# B&R Automation Studio project PLC code - cp (part 21)

#### PLC2Kernel_AutoCode.st
```iecst
// THIS CODE IS AUTOGENERATED. DO NOT MODIFY IT WITH AUTOMATION STUDIO
// Generation: 10/07/2024 16:17:34
// Program version: 2.1.4.0

ACTION PLC2Kernel_AutoCode:
HoldingRegister[1000]:=gPLC.iVarsVersion0;
HoldingRegister[1001]:=gPLC.iVarsVersion1;
HoldingRegister[1002]:=gPLC.iVarsVersion2;
HoldingRegister[1003]:=gPLC.iVersion0;
HoldingRegister[1004]:=gPLC.iVersion1;
HoldingRegister[1005]:=gPLC.iVersion2;
HoldingRegister[1006]:=gPLC.iVersion3;
HoldingRegister[1007].0:=gMachine.Al.Alarm.xAlr24Vdc;
HoldingRegister[1007].1:=gTransVacuum[1].parSw.xActiveOutOfProduction;
HoldingRegister[1007].2:=gTransVacuum[1].Status.xStartedMan;
HoldingRegister[1007].3:=gInks[1].parSw.xActTestMode;
HoldingRegister[1007].4:=gInks[2].parSw.xActTestMode;
HoldingRegister[1007].5:=gInks[3].parSw.xActTestMode;
HoldingRegister[1007].6:=gInks[4].parSw.xActTestMode;
HoldingRegister[1007].7:=gInks[5].parSw.xActTestMode;
HoldingRegister[1007].8:=gInks[6].parSw.xActTestMode;
HoldingRegister[1007].9:=gInks[7].parSw.xActTestMode;
HoldingRegister[1007].10:=gInks[8].parSw.xActTestMode;
HoldingRegister[1007].11:=gInks[9].parSw.xActTestMode;
HoldingRegister[1007].12:=gInks[10].parSw.xActTestMode;
HoldingRegister[1007].13:=gInks[11].parSw.xActTestMode;
HoldingRegister[1007].14:=gInks[12].parSw.xActTestMode;
HoldingRegister[1007].15:=gMachine.Al.Alarm.xAlarmAir1;
HoldingRegister[1008].0:=gBlock[1].Al.xAlAirVenturi;
HoldingRegister[1008].1:=gBlock[2].Al.xAlAirVenturi;
HoldingRegister[1008].2:=gMachine.Al.Alarm.xNotLoadedImage;
HoldingRegister[1008].4:=gMachine.St.Mode.xAuto;
HoldingRegister[1008].5:=gBlock[1].Al.xAlrRearSafety;
HoldingRegister[1008].6:=gBlock[2].Al.xAlrRearSafety;
HoldingRegister[1008].7:=gBlock[1].Al.xAlrDecreaseCleanOffset;
HoldingRegister[1008].8:=gBlock[2].Al.xAlrDecreaseCleanOffset;
HoldingRegister[1008].9:=gInks[1].status.xEnabledBarToPrint;
HoldingRegister[1008].10:=gInks[2].status.xEnabledBarToPrint;
HoldingRegister[1008].11:=gInks[3].status.xEnabledBarToPrint;
HoldingRegister[1008].12:=gInks[4].status.xEnabledBarToPrint;
HoldingRegister[1008].13:=gInks[5].status.xEnabledBarToPrint;
HoldingRegister[1008].14:=gInks[6].status.xEnabledBarToPrint;
HoldingRegister[1008].15:=gInks[7].status.xEnabledBarToPrint;
HoldingRegister[1009].0:=gInks[8].status.xEnabledBarToPrint;
HoldingRegister[1009].1:=gInks[9].status.xEnabledBarToPrint;
HoldingRegister[1009].2:=gInks[10].status.xEnabledBarToPrint;
HoldingRegister[1009].3:=gInks[11].status.xEnabledBarToPrint;
HoldingRegister[1009].4:=gInks[12].status.xEnabledBarToPrint;
HoldingRegister[1009].5:=gMachine.Al.Alarm.xAlarmNotInPrintPosition;
HoldingRegister[1009].6:=gBlock[1].Al.xAlrFrontCurtain;
HoldingRegister[1009].7:=gBlock[2].Al.xAlrFrontCurtain;
HoldingRegister[1009].10:=gBelt.Al.xControllerNotReady;
HoldingRegister[1009].11:=gThicknessCtrl.status.Belt.xBeltEmpty;
HoldingRegister[1009].13:=gBlock[1].Al.xSiUnitPowerOff;
HoldingRegister[1009].14:=gBlock[2].Al.xSiUnitPowerOff;
HoldingRegister[1009].15:=gTransVacuum[1].Alarms.xAlrVacuumSensor;
HoldingRegister[1010].0:=gTransVacuum[2].Alarms.xAlrVacuumSensor;
HoldingRegister[1010].1:=gBlock[1].Al.xAlrDriveProtection;
HoldingRegister[1010].2:=gBlock[2].Al.xAlrDriveProtection;
HoldingRegister[1010].3:=gInks[1].Al.xAlrBrokenMeniscus;
HoldingRegister[1010].4:=gInks[2].Al.xAlrBrokenMeniscus;
HoldingRegister[1010].5:=gInks[3].Al.xAlrBrokenMeniscus;
HoldingRegister[1010].6:=gInks[4].Al.xAlrBrokenMeniscus;
HoldingRegister[1010].7:=gInks[5].Al.xAlrBrokenMeniscus;
HoldingRegister[1010].8:=gInks[6].Al.xAlrBrokenMeniscus;
HoldingRegister[1010].9:=gInks[7].Al.xAlrBrokenMeniscus;
HoldingRegister[1010].10:=gInks[8].Al.xAlrBrokenMeniscus;
HoldingRegister[1010].11:=gInks[9].Al.xAlrBrokenMeniscus;
HoldingRegister[1010].12:=gInks[10].Al.xAlrBrokenMeniscus;
HoldingRegister[1010].13:=gInks[11].Al.xAlrBrokenMeniscus;
HoldingRegister[1010].14:=gInks[12].Al.xAlrBrokenMeniscus;
HoldingRegister[1010].15:=gChiller[1].Alarm.xCheckChiller;
HoldingRegister[1011].0:=gBlock[1].Al.xAlrCheckHomingSensor;
HoldingRegister[1011].1:=gBlock[2].Al.xAlrCheckHomingSensor;
HoldingRegister[1011].2:=gChiller[1].Alarm.xInAlarm;
HoldingRegister[1011].3:=gChiller[1].Alarm.xNotRunning;
HoldingRegister[1011].4:=gMachine.parSw.Clean.xCleaningBlocksInSeq;
HoldingRegister[1011].5:=gBlock[1].Al.xCleanMotorControllerNotReady;
HoldingRegister[1011].6:=gBlock[2].Al.xCleanMotorControllerNotReady;
HoldingRegister[1011].7:=gBelt.Al.xAlrComDrive;
HoldingRegister[1011].8:=gBlock[1].Al.xAlrComBarMtr;
HoldingRegister[1011].9:=gBlock[2].Al.xAlrComBarMtr;
HoldingRegister[1011].10:=gBlock[1].Al.xAlrComCleanMtr;
HoldingRegister[1011].11:=gBlock[2].Al.xAlrComCleanMtr;
HoldingRegister[1011].12:=gBlock[1].Al.xAlrComSiUnit;
HoldingRegister[1011].13:=gBlock[2].Al.xAlrComSiUnit;
HoldingRegister[1012].0:=gTransVacuum[1].Alarms.xAlrComsBlower;
HoldingRegister[1012].1:=gNonCrash[1].Alarms.xAlrComsDrive;
HoldingRegister[1012].2:=gTransVacuum[2].Alarms.xAlrComsBlower;
HoldingRegister[1012].3:=gMachine.Al.Alarm.xAlarmComPcPLC;
HoldingRegister[1012].4:=gPhotoCells.Alarms.xComsMotorError;
HoldingRegister[1012].7:=gMachine.St.Consent.xConsent;
HoldingRegister[1012].8:=gPhotoCells.Alarms.xContinuousActPDPhcell;
HoldingRegister[1012].9:=gMachine.Pt.xControlledByLine;
HoldingRegister[1012].10:=gBlock[1].Al.xAlrControllerNotReady;
HoldingRegister[1012].11:=gBlock[2].Al.xAlrControllerNotReady;
HoldingRegister[1012].12:=gNonCrash[1].Alarms.xControllerNotReady;
HoldingRegister[1012].13:=gBlock[1].Al.xAlrBlockReachedMaxPosition;
HoldingRegister[1012].14:=gBlock[2].Al.xAlrBlockReachedMaxPosition;
HoldingRegister[1012].15:=gInks[1].Al.xAlrTankToFillIn;
HoldingRegister[1013].0:=gInks[2].Al.xAlrTankToFillIn;
HoldingRegister[1013].1:=gInks[3].Al.xAlrTankToFillIn;
HoldingRegister[1013].2:=gInks[4].Al.xAlrTankToFillIn;
HoldingRegister[1013].3:=gInks[5].Al.xAlrTankToFillIn;
HoldingRegister[1013].4:=gInks[6].Al.xAlrTankToFillIn;
HoldingRegister[1013].5:=gInks[7].Al.xAlrTankToFillIn;
HoldingRegister[1013].6:=gInks[8].Al.xAlrTankToFillIn;
HoldingRegister[1013].7:=gInks[9].Al.xAlrTankToFillIn;
HoldingRegister[1013].8:=gInks[10].Al.xAlrTankToFillIn;
HoldingRegister[1013].9:=gInks[11].Al.xAlrTankToFillIn;
HoldingRegister[1013].10:=gInks[12].Al.xAlrTankToFillIn;
HoldingRegister[1013].11:=gInks[1].Al.xAlrTankEmpty;
HoldingRegister[1013].12:=gInks[2].Al.xAlrTankEmpty;
HoldingRegister[1013].13:=gInks[3].Al.xAlrTankEmpty;
HoldingRegister[1013].14:=gInks[4].Al.xAlrTankEmpty;
HoldingRegister[1013].15:=gInks[5].Al.xAlrTankEmpty;
HoldingRegister[1014].0:=gInks[6].Al.xAlrTankEmpty;
HoldingRegister[1014].1:=gInks[7].Al.xAlrTankEmpty;
HoldingRegister[1014].2:=gInks[8].Al.xAlrTankEmpty;
HoldingRegister[1014].3:=gInks[9].Al.xAlrTankEmpty;
HoldingRegister[1014].4:=gInks[10].Al.xAlrTankEmpty;
HoldingRegister[1014].5:=gInks[11].Al.xAlrTankEmpty;
HoldingRegister[1014].6:=gInks[12].Al.xAlrTankEmpty;
HoldingRegister[1014].7:=gInks[1].Al.xAlrDiffInCtrlTempTank;
HoldingRegister[1014].8:=gInks[2].Al.xAlrDiffInCtrlTempTank;
HoldingRegister[1014].9:=gInks[3].Al.xAlrDiffInCtrlTempTank;
HoldingRegister[1014].10:=gInks[4].Al.xAlrDiffInCtrlTempTank;
HoldingRegister[1014].11:=gInks[5].Al.xAlrDiffInCtrlTempTank;
HoldingRegister[1014].12:=gInks[6].Al.xAlrDiffInCtrlTempTank;
HoldingRegister[1014].13:=gInks[7].Al.xAlrDiffInCtrlTempTank;
HoldingRegister[1014].14:=gInks[8].Al.xAlrDiffInCtrlTempTank;
HoldingRegister[1014].15:=gInks[9].Al.xAlrDiffInCtrlTempTank;
HoldingRegister[1015].0:=gInks[10].Al.xAlrDiffInCtrlTempTank;
HoldingRegister[1015].1:=gInks[11].Al.xAlrDiffInCtrlTempTank;
HoldingRegister[1015].2:=gInks[12].Al.xAlrDiffInCtrlTempTank;
HoldingRegister[1015].3:=gInks[1].Al.xAlrDiffInCtrlTemp;
HoldingRegister[1015].4:=gInks[2].Al.xAlrDiffInCtrlTemp;
HoldingRegister[1015].5:=gInks[3].Al.xAlrDiffInCtrlTemp;
HoldingRegister[1015].6:=gInks[4].Al.xAlrDiffInCtrlTemp;
HoldingRegister[1015].7:=gInks[5].Al.xAlrDiffInCtrlTemp;
HoldingRegister[1015].8:=gInks[6].Al.xAlrDiffInCtrlTemp;
HoldingRegister[1015].9:=gInks[7].Al.xAlrDiffInCtrlTemp;
HoldingRegister[1015].10:=gInks[8].Al.xAlrDiffInCtrlTemp;
HoldingRegister[1015].11:=gInks[9].Al.xAlrDiffInCtrlTemp;
HoldingRegister[1015].12:=gInks[10].Al.xAlrDiffInCtrlTemp;
HoldingRegister[1015].13:=gInks[11].Al.xAlrDiffInCtrlTemp;
HoldingRegister[1015].14:=gInks[12].Al.xAlrDiffInCtrlTemp;
HoldingRegister[1015].15:=gBlock[1].Al.xAlrDif;
HoldingRegister[1016].0:=gBlock[2].Al.xAlrDif;
HoldingRegister[1016].2:=gNonCrash[1].Alarms.xAlrDiffContact;
HoldingRegister[1016].3:=gInks[1].Al.xAlrDifCtrlTempExcessive;
HoldingRegister[1016].4:=gInks[2].Al.xAlrDifCtrlTempExcessive;
HoldingRegister[1016].5:=gInks[3].Al.xAlrDifCtrlTempExcessive;
HoldingRegister[1016].6:=gInks[4].Al.xAlrDifCtrlTempExcessive;
HoldingRegister[1016].7:=gInks[5].Al.xAlrDifCtrlTempExcessive;
HoldingRegister[1016].8:=gInks[6].Al.xAlrDifCtrlTempExcessive;
HoldingRegister[1016].9:=gInks[7].Al.xAlrDifCtrlTempExcessive;
HoldingRegister[1016].10:=gInks[8].Al.xAlrDifCtrlTempExcessive;
HoldingRegister[1016].11:=gInks[9].Al.xAlrDifCtrlTempExcessive;
HoldingRegister[1016].12:=gInks[10].Al.xAlrDifCtrlTempExcessive;
HoldingRegister[1016].13:=gInks[11].Al.xAlrDifCtrlTempExcessive;
HoldingRegister[1016].14:=gInks[12].Al.xAlrDifCtrlTempExcessive;
HoldingRegister[1016].15:=gInks[1].Al.xAlrDiffVacuum;
HoldingRegister[1017].0:=gInks[2].Al.xAlrDiffVacuum;
HoldingRegister[1017].1:=gInks[3].Al.xAlrDiffVacuum;
HoldingRegister[1017].2:=gInks[4].Al.xAlrDiffVacuum;
HoldingRegister[1017].3:=gInks[5].Al.xAlrDiffVacuum;
HoldingRegister[1017].4:=gInks[6].Al.xAlrDiffVacuum;
HoldingRegister[1017].5:=gInks[7].Al.xAlrDiffVacuum;
HoldingRegister[1017].6:=gInks[8].Al.xAlrDiffVacuum;
HoldingRegister[1017].7:=gInks[9].Al.xAlrDiffVacuum;
HoldingRegister[1017].8:=gInks[10].Al.xAlrDiffVacuum;
HoldingRegister[1017].9:=gInks[11].Al.xAlrDiffVacuum;
HoldingRegister[1017].10:=gInks[12].Al.xAlrDiffVacuum;
HoldingRegister[1017].11:=gDing.Alarms.xAlDingNoDigLaserSensor;
HoldingRegister[1017].12:=gMachine.parSw.Dtp.xDoubleLine;
HoldingRegister[1017].13:=gMachine.St.xDoubleLineAllowed;
HoldingRegister[1017].14:=gBlock[1].Al.xAlrFrontEmergencyStop;
HoldingRegister[1017].15:=gBlock[2].Al.xAlrFrontEmergencyStop;
HoldingRegister[1018].0:=gBlock[1].Al.xAlrFrontSafetyCircuit;
HoldingRegister[1018].1:=gBlock[2].Al.xAlrFrontSafetyCircuit;
HoldingRegister[1018].2:=gBlock[1].Al.xAlrRearEmergencyStop;
HoldingRegister[1018].3:=gBlock[2].Al.xAlrRearEmergencyStop;
HoldingRegister[1018].4:=gBlock[1].Al.xAlrRearSafetyCircuit;
HoldingRegister[1018].5:=gBlock[2].Al.xAlrRearSafetyCircuit;
HoldingRegister[1018].6:=gBlock[1].Status.xIsWaterBlock;
HoldingRegister[1018].7:=gBlock[2].Status.xIsWaterBlock;
HoldingRegister[1018].9:=gJamDetect[1].Parameters.xJamEnabled;
HoldingRegister[1018].10:=gNonCrash[1].Status.xEnabled;
HoldingRegister[1018].11:=gMachine.parSw.Clean.xEnableCleaningInStopMode;
HoldingRegister[1018].12:=gBlock[1].parSw.xEnableToMovements;
HoldingRegister[1018].13:=gBlock[2].parSw.xEnableToMovements;
HoldingRegister[1018].14:=gBlock[1].Al.xAlrEnabCleanMtrDiffLvL;
HoldingRegister[1018].15:=gBlock[2].Al.xAlrEnabCleanMtrDiffLvL;
HoldingRegister[1019].0:=gInks[1].parSw.Temp.xTankHeaterEnabled;
HoldingRegister[1019].1:=gInks[2].parSw.Temp.xTankHeaterEnabled;
HoldingRegister[1019].2:=gInks[3].parSw.Temp.xTankHeaterEnabled;
HoldingRegister[1019].3:=gInks[4].parSw.Temp.xTankHeaterEnabled;
HoldingRegister[1019].4:=gInks[5].parSw.Temp.xTankHeaterEnabled;
HoldingRegister[1019].5:=gInks[6].parSw.Temp.xTankHeaterEnabled;
HoldingRegister[1019].6:=gInks[7].parSw.Temp.xTankHeaterEnabled;
HoldingRegister[1019].7:=gInks[8].parSw.Temp.xTankHeaterEnabled;
HoldingRegister[1019].8:=gInks[9].parSw.Temp.xTankHeaterEnabled;
HoldingRegister[1019].9:=gInks[10].parSw.Temp.xTankHeaterEnabled;
HoldingRegister[1019].10:=gInks[11].parSw.Temp.xTankHeaterEnabled;
HoldingRegister[1019].11:=gInks[12].parSw.Temp.xTankHeaterEnabled;
HoldingRegister[1019].12:=gBlock[1].parSw.xEnableToPrint;
HoldingRegister[1019].13:=gBlock[2].parSw.xEnableToPrint;
HoldingRegister[1019].14:=gChiller[1].Alarm.xAlrEnvTempSensBrokn;
HoldingRegister[1019].15:=gTransVacuum[1].Alarms.xAlrDriveBlowerError;
HoldingRegister[1020].0:=gNonCrash[1].Alarms.xAlrDriveError;
HoldingRegister[1020].1:=gPhotoCells.Alarms.xMotorError;
HoldingRegister[1020].2:=gTransVacuum[2].Alarms.xAlrDriveBlowerError;
HoldingRegister[1020].3:=gMachine.parSw.Electronics.xPrintServerOK;
HoldingRegister[1020].4:=gMachine.parSw.Electronics.xRobotReadyL1;
HoldingRegister[1020].5:=gMachine.parSw.Electronics.xRobotReadyL2;
HoldingRegister[1020].6:=gInks[1].Al.xAlrVacuumSensor1;
HoldingRegister[1020].7:=gInks[2].Al.xAlrVacuumSensor1;
HoldingRegister[1020].8:=gInks[3].Al.xAlrVacuumSensor1;
HoldingRegister[1020].9:=gInks[4].Al.xAlrVacuumSensor1;
HoldingRegister[1020].10:=gInks[5].Al.xAlrVacuumSensor1;
HoldingRegister[1020].11:=gInks[6].Al.xAlrVacuumSensor1;
HoldingRegister[1020].12:=gInks[7].Al.xAlrVacuumSensor1;
HoldingRegister[1020].13:=gInks[8].Al.xAlrVacuumSensor1;
HoldingRegister[1020].14:=gInks[9].Al.xAlrVacuumSensor1;
HoldingRegister[1020].15:=gInks[10].Al.xAlrVacuumSensor1;
HoldingRegister[1021].0:=gInks[11].Al.xAlrVacuumSensor1;
HoldingRegister[1021].1:=gInks[12].Al.xAlrVacuumSensor1;
HoldingRegister[1021].2:=gInks[1].Al.xAlrVacuumSensor2;
HoldingRegister[1021].3:=gInks[2].Al.xAlrVacuumSensor2;
HoldingRegister[1021].4:=gInks[3].Al.xAlrVacuumSensor2;
HoldingRegister[1021].5:=gInks[4].Al.xAlrVacuumSensor2;
HoldingRegister[1021].6:=gInks[5].Al.xAlrVacuumSensor2;
HoldingRegister[1021].7:=gInks[6].Al.xAlrVacuumSensor2;
HoldingRegister[1021].8:=gInks[7].Al.xAlrVacuumSensor2;
HoldingRegister[1021].9:=gInks[8].Al.xAlrVacuumSensor2;
HoldingRegister[1021].10:=gInks[9].Al.xAlrVacuumSensor2;
HoldingRegister[1021].11:=gInks[10].Al.xAlrVacuumSensor2;
HoldingRegister[1021].12:=gInks[11].Al.xAlrVacuumSensor2;
HoldingRegister[1021].13:=gInks[12].Al.xAlrVacuumSensor2;
HoldingRegister[1021].14:=gBelt.Al.xAlrPowerBeltError;
HoldingRegister[1021].15:=gBlock[1].Al.xAlrFrontSafety;
HoldingRegister[1022].0:=gBlock[2].Al.xAlrFrontSafety;
HoldingRegister[1022].1:=gTransVacuum[1].Alarms.xAlrJointSystemPressure;
HoldingRegister[1022].2:=gMachine.parSw.CleanBelt.xCleanBeltByTiles;
HoldingRegister[1022].3:=gMachine.parSw.CleanBelt.xCleanBeltByTime;
HoldingRegister[1022].4:=gMachine.parSw.CleanBeltTop.xCleanBeltByTiles;
HoldingRegister[1022].5:=gMachine.parSw.CleanBeltTop.xCleanBeltByTime;
HoldingRegister[1022].6:=gMachine.Al.Alarm.xAlarmEnableWithoutBarsOn;
HoldingRegister[1022].7:=gInks[1].Al.xAlrHeaterOutFault;
HoldingRegister[1022].8:=gInks[2].Al.xAlrHeaterOutFault;
HoldingRegister[1022].9:=gInks[3].Al.xAlrHeaterOutFault;
HoldingRegister[1022].10:=gInks[4].Al.xAlrHeaterOutFault;
HoldingRegister[1022].11:=gInks[5].Al.xAlrHeaterOutFault;
HoldingRegister[1022].12:=gInks[6].Al.xAlrHeaterOutFault;
HoldingRegister[1022].13:=gInks[7].Al.xAlrHeaterOutFault;
HoldingRegister[1022].14:=gInks[8].Al.xAlrHeaterOutFault;
HoldingRegister[1022].15:=gInks[9].Al.xAlrHeaterOutFault;
HoldingRegister[1023].0:=gInks[10].Al.xAlrHeaterOutFault;
HoldingRegister[1023].1:=gInks[11].Al.xAlrHeaterOutFault;
HoldingRegister[1023].2:=gInks[12].Al.xAlrHeaterOutFault;
HoldingRegister[1023].3:=gInks[1].Al.xAlrHeaterReachsMaxTemp;
HoldingRegister[1023].4:=gInks[2].Al.xAlrHeaterReachsMaxTemp;
HoldingRegister[1023].5:=gInks[3].Al.xAlrHeaterReachsMaxTemp;
HoldingRegister[1023].6:=gInks[4].Al.xAlrHeaterReachsMaxTemp;
HoldingRegister[1023].7:=gInks[5].Al.xAlrHeaterReachsMaxTemp;
HoldingRegister[1023].8:=gInks[6].Al.xAlrHeaterReachsMaxTemp;
HoldingRegister[1023].9:=gInks[7].Al.xAlrHeaterReachsMaxTemp;
HoldingRegister[1023].10:=gInks[8].Al.xAlrHeaterReachsMaxTemp;
HoldingRegister[1023].11:=gInks[9].Al.xAlrHeaterReachsMaxTemp;
HoldingRegister[1023].12:=gInks[10].Al.xAlrHeaterReachsMaxTemp;
HoldingRegister[1023].13:=gInks[11].Al.xAlrHeaterReachsMaxTemp;
HoldingRegister[1023].14:=gInks[12].Al.xAlrHeaterReachsMaxTemp;
HoldingRegister[1023].15:=gInks[1].Al.xAlrHeaterTankReachsMaxTemp;
HoldingRegister[1024].0:=gInks[2].Al.xAlrHeaterTankReachsMaxTemp;
HoldingRegister[1024].1:=gInks[3].Al.xAlrHeaterTankReachsMaxTemp;
HoldingRegister[1024].2:=gInks[4].Al.xAlrHeaterTankReachsMaxTemp;
HoldingRegister[1024].3:=gInks[5].Al.xAlrHeaterTankReachsMaxTemp;
HoldingRegister[1024].4:=gInks[6].Al.xAlrHeaterTankReachsMaxTemp;
HoldingRegister[1024].5:=gInks[7].Al.xAlrHeaterTankReachsMaxTemp;
HoldingRegister[1024].6:=gInks[8].Al.xAlrHeaterTankReachsMaxTemp;
HoldingRegister[1024].7:=gInks[9].Al.xAlrHeaterTankReachsMaxTemp;
HoldingRegister[1024].8:=gInks[10].Al.xAlrHeaterTankReachsMaxTemp;
HoldingRegister[1024].9:=gInks[11].Al.xAlrHeaterTankReachsMaxTemp;
HoldingRegister[1024].10:=gInks[12].Al.xAlrHeaterTankReachsMaxTemp;
HoldingRegister[1024].11:=gBelt.Al.xAlrProtDrive;
HoldingRegister[1024].12:=gBlock[1].Al.xAlrCleanMtrNoRef;
HoldingRegister[1024].13:=gBlock[2].Al.xAlrCleanMtrNoRef;
HoldingRegister[1024].14:=gBlock[1].Status.Icla.xHomed;
HoldingRegister[1024].15:=gBlock[2].Status.Icla.xHomed;
HoldingRegister[1025].0:=gMachine.Al.Warning.xNotLoadedImage;
HoldingRegister[1025].1:=gInks[1].Al.xAlrLevelSensorError;
HoldingRegister[1025].2:=gInks[2].Al.xAlrLevelSensorError;
HoldingRegister[1025].3:=gInks[3].Al.xAlrLevelSensorError;
HoldingRegister[1025].4:=gInks[4].Al.xAlrLevelSensorError;
HoldingRegister[1025].5:=gInks[5].Al.xAlrLevelSensorError;
HoldingRegister[1025].6:=gInks[6].Al.xAlrLevelSensorError;
HoldingRegister[1025].7:=gInks[7].Al.xAlrLevelSensorError;
HoldingRegister[1025].8:=gInks[8].Al.xAlrLevelSensorError;
HoldingRegister[1025].9:=gInks[9].Al.xAlrLevelSensorError;
HoldingRegister[1025].10:=gInks[10].Al.xAlrLevelSensorError;
HoldingRegister[1025].11:=gInks[11].Al.xAlrLevelSensorError;
HoldingRegister[1025].12:=gInks[12].Al.xAlrLevelSensorError;
HoldingRegister[1025].13:=gInks[1].Al.xAlrIncoherTempHeat;
HoldingRegister[1025].14:=gInks[2].Al.xAlrIncoherTempHeat;
HoldingRegister[1025].15:=gInks[3].Al.xAlrIncoherTempHeat;
HoldingRegister[1026].0:=gInks[4].Al.xAlrIncoherTempHeat;
HoldingRegister[1026].1:=gInks[5].Al.xAlrIncoherTempHeat;
HoldingRegister[1026].2:=gInks[6].Al.xAlrIncoherTempHeat;
HoldingRegister[1026].3:=gInks[7].Al.xAlrIncoherTempHeat;
HoldingRegister[1026].4:=gInks[8].Al.xAlrIncoherTempHeat;
HoldingRegister[1026].5:=gInks[9].Al.xAlrIncoherTempHeat;
HoldingRegister[1026].6:=gInks[10].Al.xAlrIncoherTempHeat;
HoldingRegister[1026].7:=gInks[11].Al.xAlrIncoherTempHeat;
HoldingRegister[1026].8:=gInks[12].Al.xAlrIncoherTempHeat;
HoldingRegister[1026].9:=gPhotoCells.Alarms.xIncoherPhotocellSystem;
HoldingRegister[1026].10:=gBlock[1].Al.xAlrIncoherPositCleanMtr;
HoldingRegister[1026].11:=gBlock[2].Al.xAlrIncoherPositCleanMtr;
HoldingRegister[1026].12:=gInks[1].Al.xAlrIncoherTempTank;
HoldingRegister[1026].13:=gInks[2].Al.xAlrIncoherTempTank;
HoldingRegister[1026].14:=gInks[3].Al.xAlrIncoherTempTank;
HoldingRegister[1026].15:=gInks[4].Al.xAlrIncoherTempTank;
HoldingRegister[1027].0:=gInks[5].Al.xAlrIncoherTempTank;
HoldingRegister[1027].1:=gInks[6].Al.xAlrIncoherTempTank;
HoldingRegister[1027].2:=gInks[7].Al.xAlrIncoherTempTank;
HoldingRegister[1027].3:=gInks[8].Al.xAlrIncoherTempTank;
HoldingRegister[1027].4:=gInks[9].Al.xAlrIncoherTempTank;
HoldingRegister[1027].5:=gInks[10].Al.xAlrIncoherTempTank;
HoldingRegister[1027].6:=gInks[11].Al.xAlrIncoherTempTank;
HoldingRegister[1027].7:=gInks[12].Al.xAlrIncoherTempTank;
HoldingRegister[1027].8:=gMachine.commands.xCompenserLine1;
HoldingRegister[1027].9:=gMachine.commands.xCompenserLine2;
HoldingRegister[1027].10:=gNonCrash[1].Status.xInstalled;
HoldingRegister[1027].11:=gJamPerInk[1].xAlrJamCrash;
HoldingRegister[1027].12:=gJamPerInk[2].xAlrJamCrash;
HoldingRegister[1027].13:=gJamPerInk[3].xAlrJamCrash;
HoldingRegister[1027].14:=gJamPerInk[4].xAlrJamCrash;
HoldingRegister[1027].15:=gJamPerInk[5].xAlrJamCrash;
HoldingRegister[1028].0:=gJamPerInk[6].xAlrJamCrash;
HoldingRegister[1028].1:=gJamPerInk[7].xAlrJamCrash;
HoldingRegister[1028].2:=gJamPerInk[8].xAlrJamCrash;
HoldingRegister[1028].3:=gJamPerInk[9].xAlrJamCrash;
HoldingRegister[1028].4:=gJamPerInk[10].xAlrJamCrash;
HoldingRegister[1028].5:=gJamPerInk[11].xAlrJamCrash;
HoldingRegister[1028].6:=gJamPerInk[12].xAlrJamCrash;
HoldingRegister[1028].7:=gJamPerInk[1].xAlrJamTest;
HoldingRegister[1028].8:=gJamPerInk[2].xAlrJamTest;
HoldingRegister[1028].9:=gJamPerInk[3].xAlrJamTest;
HoldingRegister[1028].10:=gJamPerInk[4].xAlrJamTest;
HoldingRegister[1028].11:=gJamPerInk[5].xAlrJamTest;
HoldingRegister[1028].12:=gJamPerInk[6].xAlrJamTest;
HoldingRegister[1028].13:=gJamPerInk[7].xAlrJamTest;
HoldingRegister[1028].14:=gJamPerInk[8].xAlrJamTest;
HoldingRegister[1028].15:=gJamPerInk[9].xAlrJamTest;
HoldingRegister[1029].0:=gJamPerInk[10].xAlrJamTest;
HoldingRegister[1029].1:=gJamPerInk[11].xAlrJamTest;
HoldingRegister[1029].2:=gJamPerInk[12].xAlrJamTest;
HoldingRegister[1029].3:=gInks[1].Al.xAlrKlixonTriggered;
HoldingRegister[1029].4:=gInks[2].Al.xAlrKlixonTriggered;
HoldingRegister[1029].5:=gInks[3].Al.xAlrKlixonTriggered;
HoldingRegister[1029].6:=gInks[4].Al.xAlrKlixonTriggered;
HoldingRegister[1029].7:=gInks[5].Al.xAlrKlixonTriggered;
HoldingRegister[1029].8:=gInks[6].Al.xAlrKlixonTriggered;
HoldingRegister[1029].9:=gInks[7].Al.xAlrKlixonTriggered;
HoldingRegister[1029].10:=gInks[8].Al.xAlrKlixonTriggered;
HoldingRegister[1029].11:=gInks[9].Al.xAlrKlixonTriggered;
HoldingRegister[1029].12:=gInks[10].Al.xAlrKlixonTriggered;
HoldingRegister[1029].13:=gInks[11].Al.xAlrKlixonTriggered;
HoldingRegister[1029].14:=gInks[12].Al.xAlrKlixonTriggered;
HoldingRegister[1029].15:=gMachine.St.Consent.xLackOfConsent;
HoldingRegister[1030].0:=gDing.Alarms.xAlDingNotReferenced;
HoldingRegister[1030].1:=gMachine.parSw.CleanBelt.xCleanBeltContinue;
HoldingRegister[1030].2:=gMachine.parSw.CleanBeltTop.xCleanBeltContinue;
HoldingRegister[1030].3:=gMachine.Al.Warning.xExternalCleanActive;
HoldingRegister[1030].4:=gBlock[1].Al.xAlCleanInterrupt;
HoldingRegister[1030].5:=gBlock[2].Al.xAlCleanInterrupt;
HoldingRegister[1030].6:=gMachine.parSw.Clean.xCleanSystemByPieces;
HoldingRegister[1030].7:=gMachine.parSw.Clean.xCleanSystemByTime;
HoldingRegister[1030].8:=gMachine.St.HwData.xIsCubik;
HoldingRegister[1030].9:=gMachine.St.HwData.xIsPlatform5;
HoldingRegister[1030].10:=gMachine.St.HwData.xIsWater;
HoldingRegister[1030].12:=gMachine.parSw.PCs.xKeepPcsOn;
HoldingRegister[1030].13:=gMachine.St.Mode.xManual;
HoldingRegister[1030].14:=gMachine.St.AutoMode.xPause;
HoldingRegister[1030].15:=gInks[1].Al.xAlrInksRunnig;
HoldingRegister[1031].0:=gInks[2].Al.xAlrInksRunnig;
HoldingRegister[1031].1:=gInks[3].Al.xAlrInksRunnig;
HoldingRegister[1031].2:=gInks[4].Al.xAlrInksRunnig;
HoldingRegister[1031].3:=gInks[5].Al.xAlrInksRunnig;
HoldingRegister[1031].4:=gInks[6].Al.xAlrInksRunnig;
HoldingRegister[1031].5:=gInks[7].Al.xAlrInksRunnig;
HoldingRegister[1031].6:=gInks[8].Al.xAlrInksRunnig;
HoldingRegister[1031].7:=gInks[9].Al.xAlrInksRunnig;
HoldingRegister[1031].8:=gInks[10].Al.xAlrInksRunnig;
HoldingRegister[1031].9:=gInks[11].Al.xAlrInksRunnig;
HoldingRegister[1031].10:=gInks[12].Al.xAlrInksRunnig;
HoldingRegister[1031].11:=gThicknessCtrl.status.MediaPosition.xMediaToRejectInside;
HoldingRegister[1031].12:=gBelt.Al.xAnyDriveAlarm;
HoldingRegister[1031].13:=gBlock[1].Al.xAnyVerticalDriveAlarm;
HoldingRegister[1031].14:=gBlock[2].Al.xAnyVerticalDriveAlarm;
HoldingRegister[1031].15:=gBlock[1].Al.xAlBarMotorPowerOff;
HoldingRegister[1032].0:=gBlock[2].Al.xAlBarMotorPowerOff;
HoldingRegister[1032].1:=gBlock[1].Al.xAlrCleanMotor;
HoldingRegister[1032].2:=gBlock[2].Al.xAlrCleanMotor;
HoldingRegister[1032].5:=gInks[1].status.Tank.xMaxLevel;
HoldingRegister[1032].6:=gInks[2].status.Tank.xMaxLevel;
HoldingRegister[1032].7:=gInks[3].status.Tank.xMaxLevel;
HoldingRegister[1032].8:=gInks[4].status.Tank.xMaxLevel;
HoldingRegister[1032].9:=gInks[5].status.Tank.xMaxLevel;
HoldingRegister[1032].10:=gInks[6].status.Tank.xMaxLevel;
HoldingRegister[1032].11:=gInks[7].status.Tank.xMaxLevel;
HoldingRegister[1032].12:=gInks[8].status.Tank.xMaxLevel;
HoldingRegister[1032].13:=gInks[9].status.Tank.xMaxLevel;
HoldingRegister[1032].14:=gInks[10].status.Tank.xMaxLevel;
HoldingRegister[1032].15:=gInks[11].status.Tank.xMaxLevel;
HoldingRegister[1033].0:=gInks[12].status.Tank.xMaxLevel;
HoldingRegister[1033].1:=gInks[1].status.Tank.xMinLevel;
HoldingRegister[1033].2:=gInks[2].status.Tank.xMinLevel;
HoldingRegister[1033].3:=gInks[3].status.Tank.xMinLevel;
HoldingRegister[1033].4:=gInks[4].status.Tank.xMinLevel;
HoldingRegister[1033].5:=gInks[5].status.Tank.xMinLevel;
HoldingRegister[1033].6:=gInks[6].status.Tank.xMinLevel;
HoldingRegister[1033].7:=gInks[7].status.Tank.xMinLevel;
HoldingRegister[1033].8:=gInks[8].status.Tank.xMinLevel;
HoldingRegister[1033].9:=gInks[9].status.Tank.xMinLevel;
HoldingRegister[1033].10:=gInks[10].status.Tank.xMinLevel;
HoldingRegister[1033].11:=gInks[11].status.Tank.xMinLevel;
HoldingRegister[1033].12:=gInks[12].status.Tank.xMinLevel;
HoldingRegister[1033].13:=gMachine.Al.Alarm.xNoActionDangerCollision;
HoldingRegister[1033].14:=gMachine.Al.Alarm.xNoActionAlarmExist;
HoldingRegister[1033].15:=gPhotoCells.Alarms.xNoDigSignalLaserSensor;
HoldingRegister[1034].0:=gNonCrash[1].Alarms.xAlrOvertorque;
HoldingRegister[1034].1:=gDing.Alarms.xAlNoDingDetect;
HoldingRegister[1034].2:=gBlock[1].Al.xAlrWaterPumpPresure;
HoldingRegister[1034].3:=gBlock[2].Al.xAlrWaterPumpPresure;
HoldingRegister[1034].4:=gBelt.Al.xAxisLengthNotDefined;
HoldingRegister[1034].9:=gBlock[1].Al.xModuleTemp01;
HoldingRegister[1034].10:=gBlock[2].Al.xModuleTemp01;
HoldingRegister[1034].11:=gBlock[1].Al.xModuleTemp02;
HoldingRegister[1034].12:=gBlock[2].Al.xModuleTemp02;
HoldingRegister[1034].13:=gBlock[1].Al.xModuleTemp03;
HoldingRegister[1034].14:=gBlock[2].Al.xModuleTemp03;
HoldingRegister[1035].11:=gBelt.Al.xGearBoxNotDefined;
HoldingRegister[1035].12:=gNonCrash[1].Alarms.xGearBoxNotDefined;
HoldingRegister[1035].13:=gPhotoCells.Alarms.xNotReferenced;
HoldingRegister[1035].14:=gInks[1].Al.xAlrNoInkNoCleanManif;
HoldingRegister[1035].15:=gInks[2].Al.xAlrNoInkNoCleanManif;
HoldingRegister[1036].0:=gInks[3].Al.xAlrNoInkNoCleanManif;
HoldingRegister[1036].1:=gInks[4].Al.xAlrNoInkNoCleanManif;
HoldingRegister[1036].2:=gInks[5].Al.xAlrNoInkNoCleanManif;
HoldingRegister[1036].3:=gInks[6].Al.xAlrNoInkNoCleanManif;
HoldingRegister[1036].4:=gInks[7].Al.xAlrNoInkNoCleanManif;
HoldingRegister[1036].5:=gInks[8].Al.xAlrNoInkNoCleanManif;
HoldingRegister[1036].6:=gInks[9].Al.xAlrNoInkNoCleanManif;
HoldingRegister[1036].7:=gInks[10].Al.xAlrNoInkNoCleanManif;
HoldingRegister[1036].8:=gInks[11].Al.xAlrNoInkNoCleanManif;
HoldingRegister[1036].9:=gInks[12].Al.xAlrNoInkNoCleanManif;
HoldingRegister[1036].10:=gNonCrash[1].Alarms.xPerimeterNotDefined;
HoldingRegister[1036].11:=gMachine.Al.Warning.xMaxMovsBentTile;
HoldingRegister[1036].12:=gInks[1].parSw.xOnReverseCapped;
HoldingRegister[1036].13:=gInks[2].parSw.xOnReverseCapped;
HoldingRegister[1036].14:=gInks[3].parSw.xOnReverseCapped;
HoldingRegister[1036].15:=gInks[4].parSw.xOnReverseCapped;
HoldingRegister[1037].0:=gInks[5].parSw.xOnReverseCapped;
HoldingRegister[1037].1:=gInks[6].parSw.xOnReverseCapped;
HoldingRegister[1037].2:=gInks[7].parSw.xOnReverseCapped;
HoldingRegister[1037].3:=gInks[8].parSw.xOnReverseCapped;
HoldingRegister[1037].4:=gInks[9].parSw.xOnReverseCapped;
HoldingRegister[1037].5:=gInks[10].parSw.xOnReverseCapped;
HoldingRegister[1037].6:=gInks[11].parSw.xOnReverseCapped;
HoldingRegister[1037].7:=gInks[12].parSw.xOnReverseCapped;
HoldingRegister[1037].8:=gInks[1].parSw.xOnReverseCleaning;
HoldingRegister[1037].9:=gInks[2].parSw.xOnReverseCleaning;
HoldingRegister[1037].10:=gInks[3].parSw.xOnReverseCleaning;
HoldingRegister[1037].11:=gInks[4].parSw.xOnReverseCleaning;
HoldingRegister[1037].12:=gInks[5].parSw.xOnReverseCleaning;
HoldingRegister[1037].13:=gInks[6].parSw.xOnReverseCleaning;
HoldingRegister[1037].14:=gInks[7].parSw.xOnReverseCleaning;
HoldingRegister[1037].15:=gInks[8].parSw.xOnReverseCleaning;
HoldingRegister[1038].0:=gInks[9].parSw.xOnReverseCleaning;
HoldingRegister[1038].1:=gInks[10].parSw.xOnReverseCleaning;
HoldingRegister[1038].2:=gInks[11].parSw.xOnReverseCleaning;
HoldingRegister[1038].3:=gInks[12].parSw.xOnReverseCleaning;
HoldingRegister[1038].4:=gBlock[1].In.xTrayIn;
HoldingRegister[1038].5:=gBlock[2].In.xTrayIn;
HoldingRegister[1038].6:=gBlock[1].In.xTrayOut;
HoldingRegister[1038].7:=gBlock[2].In.xTrayOut;
HoldingRegister[1038].8:=gInks[1].signals.out.xOutPowPrintHead;
HoldingRegister[1038].9:=gInks[2].signals.out.xOutPowPrintHead;
HoldingRegister[1038].10:=gInks[3].signals.out.xOutPowPrintHead;
HoldingRegister[1038].11:=gInks[4].signals.out.xOutPowPrintHead;
HoldingRegister[1038].12:=gInks[5].signals.out.xOutPowPrintHead;
HoldingRegister[1038].13:=gInks[6].signals.out.xOutPowPrintHead;
HoldingRegister[1038].14:=gInks[7].signals.out.xOutPowPrintHead;
HoldingRegister[1038].15:=gInks[8].signals.out.xOutPowPrintHead;
HoldingRegister[1039].0:=gInks[9].signals.out.xOutPowPrintHead;
HoldingRegister[1039].1:=gInks[10].signals.out.xOutPowPrintHead;
HoldingRegister[1039].2:=gInks[11].signals.out.xOutPowPrintHead;
HoldingRegister[1039].3:=gInks[12].signals.out.xOutPowPrintHead;
HoldingRegister[1039].4:=gBlock[1].Al.xBarDriverTemp;
HoldingRegister[1039].5:=gBlock[2].Al.xBarDriverTemp;
HoldingRegister[1039].6:=gBlock[1].Al.xBarMotorTemp;
HoldingRegister[1039].7:=gBlock[2].Al.xBarMotorTemp;
HoldingRegister[1039].8:=gBelt.Al.xBeltDriverTemp;
HoldingRegister[1039].9:=gBelt.Al.xBeltMotorTemp;
HoldingRegister[1039].10:=gMachine.Al.Warning.xPCCabineSensAlrm;
HoldingRegister[1039].11:=gBelt.Al.xWrnOverTorq;
HoldingRegister[1039].12:=gMachine.Al.Alarm.xAlarmMountedPiece;
HoldingRegister[1039].13:=gInks[1].Al.xAlrStopRecircNoInk;
HoldingRegister[1039].14:=gInks[2].Al.xAlrStopRecircNoInk;
HoldingRegister[1039].15:=gInks[3].Al.xAlrStopRecircNoInk;
HoldingRegister[1040].0:=gInks[4].Al.xAlrStopRecircNoInk;
HoldingRegister[1040].1:=gInks[5].Al.xAlrStopRecircNoInk;
HoldingRegister[1040].2:=gInks[6].Al.xAlrStopRecircNoInk;
HoldingRegister[1040].3:=gInks[7].Al.xAlrStopRecircNoInk;
HoldingRegister[1040].4:=gInks[8].Al.xAlrStopRecircNoInk;
HoldingRegister[1040].5:=gInks[9].Al.xAlrStopRecircNoInk;
HoldingRegister[1040].6:=gInks[10].Al.xAlrStopRecircNoInk;
HoldingRegister[1040].7:=gInks[11].Al.xAlrStopRecircNoInk;
HoldingRegister[1040].8:=gInks[12].Al.xAlrStopRecircNoInk;
HoldingRegister[1040].9:=gMachine.St.xWorkingAsPBF;
HoldingRegister[1040].10:=gMachine.Al.Warning.xPbfCardNotOK;
HoldingRegister[1040].11:=gMachine.Al.Alarm.xPDBrokenSensorL1;
HoldingRegister[1040].12:=gMachine.Al.Alarm.xPDBrokenSensorL2;
HoldingRegister[1040].13:=gDing.Alarms.xAlDingConexionError;
HoldingRegister[1040].14:=gDing.In.xDingHigh;
HoldingRegister[1040].15:=gDing.State.xDingLowPieceDetect;
HoldingRegister[1041].0:=gPhotoCells.Inputs.Signals.xPhotoCells[1];
HoldingRegister[1041].1:=gPhotoCells.Inputs.Signals.xPhotoCells[2];
HoldingRegister[1041].2:=gPhotoCells.Inputs.Signals.xPhotoCells[3];
HoldingRegister[1041].3:=gPhotoCells.status.xMotorError;
HoldingRegister[1041].4:=gPhotoCells.status.xReferenced;
HoldingRegister[1041].5:=gBlock[1].Al.xAlrPHPowerSupply;
HoldingRegister[1041].6:=gBlock[2].Al.xAlrPHPowerSupply;
HoldingRegister[1041].7:=gMachine.Al.Alarm.xAlarmPlarformInc;
HoldingRegister[1041].10:=gMachine.Al.Alarm.xHeaterTankPsu;
HoldingRegister[1041].11:=gInks[1].Al.xAlrPrintHeadPsuFailure;
HoldingRegister[1041].12:=gInks[2].Al.xAlrPrintHeadPsuFailure;
HoldingRegister[1041].13:=gInks[3].Al.xAlrPrintHeadPsuFailure;
HoldingRegister[1041].14:=gInks[4].Al.xAlrPrintHeadPsuFailure;
HoldingRegister[1041].15:=gInks[5].Al.xAlrPrintHeadPsuFailure;
HoldingRegister[1042].0:=gInks[6].Al.xAlrPrintHeadPsuFailure;
HoldingRegister[1042].1:=gInks[7].Al.xAlrPrintHeadPsuFailure;
HoldingRegister[1042].2:=gInks[8].Al.xAlrPrintHeadPsuFailure;
HoldingRegister[1042].3:=gInks[9].Al.xAlrPrintHeadPsuFailure;
HoldingRegister[1042].4:=gInks[10].Al.xAlrPrintHeadPsuFailure;
HoldingRegister[1042].5:=gInks[11].Al.xAlrPrintHeadPsuFailure;
HoldingRegister[1042].6:=gInks[12].Al.xAlrPrintHeadPsuFailure;
HoldingRegister[1042].7:=gInks[1].Al.xAlrPrintHeadsChillerStopped;
HoldingRegister[1042].8:=gInks[2].Al.xAlrPrintHeadsChillerStopped;
HoldingRegister[1042].9:=gInks[3].Al.xAlrPrintHeadsChillerStopped;
HoldingRegister[1042].10:=gInks[4].Al.xAlrPrintHeadsChillerStopped;
HoldingRegister[1042].11:=gInks[5].Al.xAlrPrintHeadsChillerStopped;
HoldingRegister[1042].12:=gInks[6].Al.xAlrPrintHeadsChillerStopped;
HoldingRegister[1042].13:=gInks[7].Al.xAlrPrintHeadsChillerStopped;
HoldingRegister[1042].14:=gInks[8].Al.xAlrPrintHeadsChillerStopped;
HoldingRegister[1042].15:=gInks[9].Al.xAlrPrintHeadsChillerStopped;
HoldingRegister[1043].0:=gInks[10].Al.xAlrPrintHeadsChillerStopped;
HoldingRegister[1043].1:=gInks[11].Al.xAlrPrintHeadsChillerStopped;
HoldingRegister[1043].2:=gInks[12].Al.xAlrPrintHeadsChillerStopped;
HoldingRegister[1043].3:=gInks[1].Al.xAlrPumpsDCError;
HoldingRegister[1043].4:=gInks[2].Al.xAlrPumpsDCError;
HoldingRegister[1043].5:=gInks[3].Al.xAlrPumpsDCError;
HoldingRegister[1043].6:=gInks[4].Al.xAlrPumpsDCError;
HoldingRegister[1043].7:=gInks[5].Al.xAlrPumpsDCError;
HoldingRegister[1043].8:=gInks[6].Al.xAlrPumpsDCError;
HoldingRegister[1043].9:=gInks[7].Al.xAlrPumpsDCError;
HoldingRegister[1043].10:=gInks[8].Al.xAlrPumpsDCError;
HoldingRegister[1043].11:=gInks[9].Al.xAlrPumpsDCError;
HoldingRegister[1043].12:=gInks[10].Al.xAlrPumpsDCError;
HoldingRegister[1043].13:=gInks[11].Al.xAlrPumpsDCError;
HoldingRegister[1043].14:=gInks[12].Al.xAlrPumpsDCError;
HoldingRegister[1043].15:=gTransVacuum[2].Alarms.xAlrJointSystemPressure;
HoldingRegister[1044].12:=gBlock[1].Status.Motor.xBarsHoming;
HoldingRegister[1044].13:=gBlock[2].Status.Motor.xBarsHoming;
HoldingRegister[1044].14:=gBlock[1].Status.Icla.xHoming;
HoldingRegister[1044].15:=gBlock[2].Status.Icla.xHoming;
HoldingRegister[1045].0:=gPhotoCells.status.xReferencing;
HoldingRegister[1045].1:=gMachine.parSw.Shot.xRepetitionShotLine1;
HoldingRegister[1045].2:=gMachine.parSw.Shot.xRepetitionShotLine2;
HoldingRegister[1045].3:=gInks[1].status.Reverse.xReverseMan;
HoldingRegister[1045].4:=gInks[2].status.Reverse.xReverseMan;
HoldingRegister[1045].5:=gInks[3].status.Reverse.xReverseMan;
HoldingRegister[1045].6:=gInks[4].status.Reverse.xReverseMan;
HoldingRegister[1045].7:=gInks[5].status.Reverse.xReverseMan;
HoldingRegister[1045].8:=gInks[6].status.Reverse.xReverseMan;
HoldingRegister[1045].9:=gInks[7].status.Reverse.xReverseMan;
HoldingRegister[1045].10:=gInks[8].status.Reverse.xReverseMan;
HoldingRegister[1045].11:=gInks[9].status.Reverse.xReverseMan;
HoldingRegister[1045].12:=gInks[10].status.Reverse.xReverseMan;
HoldingRegister[1045].13:=gInks[11].status.Reverse.xReverseMan;
HoldingRegister[1045].14:=gInks[12].status.Reverse.xReverseMan;
HoldingRegister[1046].0:=gBlock[1].Al.xAlrTraySensor;
HoldingRegister[1046].1:=gBlock[2].Al.xAlrTraySensor;
HoldingRegister[1046].2:=gBlock[1].Al.xAlrCleanSensor;
HoldingRegister[1046].3:=gBlock[2].Al.xAlrCleanSensor;
HoldingRegister[1046].4:=gDing.Alarms.xAlDingDetect;
HoldingRegister[1046].5:=gBlock[1].Al.xAlrReferenceIncoherence;
HoldingRegister[1046].6:=gBlock[2].Al.xAlrReferenceIncoherence;
HoldingRegister[1046].7:=gBlock[1].In.xIclaSensor;
HoldingRegister[1046].8:=gBlock[2].In.xIclaSensor;
HoldingRegister[1046].9:=gBlock[1].Al.xAlrBarMtrNoRef;
HoldingRegister[1046].10:=gBlock[2].Al.xAlrBarMtrNoRef;
HoldingRegister[1046].11:=gBlock[1].Status.Motor.xBarsHomed;
HoldingRegister[1046].12:=gBlock[2].Status.Motor.xBarsHomed;
HoldingRegister[1046].13:=gMachine.Al.xAlrSafetySystemEStop;
HoldingRegister[1046].15:=gInks[1].Al.xAlrNoRecirculation;
HoldingRegister[1047].0:=gInks[2].Al.xAlrNoRecirculation;
HoldingRegister[1047].1:=gInks[3].Al.xAlrNoRecirculation;
HoldingRegister[1047].2:=gInks[4].Al.xAlrNoRecirculation;
HoldingRegister[1047].3:=gInks[5].Al.xAlrNoRecirculation;
HoldingRegister[1047].4:=gInks[6].Al.xAlrNoRecirculation;
HoldingRegister[1047].5:=gInks[7].Al.xAlrNoRecirculation;
HoldingRegister[1047].6:=gInks[8].Al.xAlrNoRecirculation;
HoldingRegister[1047].7:=gInks[9].Al.xAlrNoRecirculation;
HoldingRegister[1047].8:=gInks[10].Al.xAlrNoRecirculation;
HoldingRegister[1047].9:=gInks[11].Al.xAlrNoRecirculation;
HoldingRegister[1047].10:=gInks[12].Al.xAlrNoRecirculation;
HoldingRegister[1047].11:=gInks[1].Al.xAlrNoRecircStop;
HoldingRegister[1047].12:=gInks[2].Al.xAlrNoRecircStop;
HoldingRegister[1047].13:=gInks[3].Al.xAlrNoRecircStop;
HoldingRegister[1047].14:=gInks[4].Al.xAlrNoRecircStop;
HoldingRegister[1047].15:=gInks[5].Al.xAlrNoRecircStop;
HoldingRegister[1048].0:=gInks[6].Al.xAlrNoRecircStop;
HoldingRegister[1048].1:=gInks[7].Al.xAlrNoRecircStop;
HoldingRegister[1048].2:=gInks[8].Al.xAlrNoRecircStop;
HoldingRegister[1048].3:=gInks[9].Al.xAlrNoRecircStop;
HoldingRegister[1048].4:=gInks[10].Al.xAlrNoRecircStop;
HoldingRegister[1048].5:=gInks[11].Al.xAlrNoRecircStop;
HoldingRegister[1048].6:=gInks[12].Al.xAlrNoRecircStop;
HoldingRegister[1048].7:=gBelt.Al.xAlrOverTorque;
HoldingRegister[1048].10:=gInks[1].Al.xAlrOverPressure;
HoldingRegister[1048].11:=gInks[2].Al.xAlrOverPressure;
HoldingRegister[1048].12:=gInks[3].Al.xAlrOverPressure;
HoldingRegister[1048].13:=gInks[4].Al.xAlrOverPressure;
HoldingRegister[1048].14:=gInks[5].Al.xAlrOverPressure;
HoldingRegister[1048].15:=gInks[6].Al.xAlrOverPressure;
HoldingRegister[1049].0:=gInks[7].Al.xAlrOverPressure;
HoldingRegister[1049].1:=gInks[8].Al.xAlrOverPressure;
HoldingRegister[1049].2:=gInks[9].Al.xAlrOverPressure;
HoldingRegister[1049].3:=gInks[10].Al.xAlrOverPressure;
HoldingRegister[1049].4:=gInks[11].Al.xAlrOverPressure;
HoldingRegister[1049].5:=gInks[12].Al.xAlrOverPressure;
HoldingRegister[1049].6:=gInks[1].Al.xAlrTempSensor;
HoldingRegister[1049].7:=gInks[2].Al.xAlrTempSensor;
HoldingRegister[1049].8:=gInks[3].Al.xAlrTempSensor;
HoldingRegister[1049].9:=gInks[4].Al.xAlrTempSensor;
HoldingRegister[1049].10:=gInks[5].Al.xAlrTempSensor;
HoldingRegister[1049].11:=gInks[6].Al.xAlrTempSensor;
HoldingRegister[1049].12:=gInks[7].Al.xAlrTempSensor;
HoldingRegister[1049].13:=gInks[8].Al.xAlrTempSensor;
HoldingRegister[1049].14:=gInks[9].Al.xAlrTempSensor;
HoldingRegister[1049].15:=gInks[10].Al.xAlrTempSensor;
HoldingRegister[1050].0:=gInks[11].Al.xAlrTempSensor;
HoldingRegister[1050].1:=gInks[12].Al.xAlrTempSensor;
HoldingRegister[1050].2:=gInks[1].Al.xAlrVacuum1;
HoldingRegister[1050].3:=gInks[2].Al.xAlrVacuum1;
HoldingRegister[1050].4:=gInks[3].Al.xAlrVacuum1;
HoldingRegister[1050].5:=gInks[4].Al.xAlrVacuum1;
HoldingRegister[1050].6:=gInks[5].Al.xAlrVacuum1;
HoldingRegister[1050].7:=gInks[6].Al.xAlrVacuum1;
HoldingRegister[1050].8:=gInks[7].Al.xAlrVacuum1;
HoldingRegister[1050].9:=gInks[8].Al.xAlrVacuum1;
HoldingRegister[1050].10:=gInks[9].Al.xAlrVacuum1;
HoldingRegister[1050].11:=gInks[10].Al.xAlrVacuum1;
HoldingRegister[1050].12:=gInks[11].Al.xAlrVacuum1;
HoldingRegister[1050].13:=gInks[12].Al.xAlrVacuum1;
HoldingRegister[1050].14:=gInks[1].Al.xAlrVacuum2;
HoldingRegister[1050].15:=gInks[2].Al.xAlrVacuum2;
HoldingRegister[1051].0:=gInks[3].Al.xAlrVacuum2;
HoldingRegister[1051].1:=gInks[4].Al.xAlrVacuum2;
HoldingRegister[1051].2:=gInks[5].Al.xAlrVacuum2;
HoldingRegister[1051].3:=gInks[6].Al.xAlrVacuum2;
HoldingRegister[1051].4:=gInks[7].Al.xAlrVacuum2;
HoldingRegister[1051].5:=gInks[8].Al.xAlrVacuum2;
HoldingRegister[1051].6:=gInks[9].Al.xAlrVacuum2;
HoldingRegister[1051].7:=gInks[10].Al.xAlrVacuum2;
HoldingRegister[1051].8:=gInks[11].Al.xAlrVacuum2;
HoldingRegister[1051].9:=gInks[12].Al.xAlrVacuum2;
HoldingRegister[1051].10:=gMachine.Al.Warning.xMediaStoppedInside;
HoldingRegister[1051].11:=gMachine.Al.Warning.xUpNotConsent;
HoldingRegister[1051].12:=gMachine.Al.Warning.xBentTile;
HoldingRegister[1051].13:=gInks[1].Al.xAlrTankCloseToEmpty;
HoldingRegister[1051].14:=gInks[2].Al.xAlrTankCloseToEmpty;
HoldingRegister[1051].15:=gInks[3].Al.xAlrTankCloseToEmpty;
HoldingRegister[1052].0:=gInks[4].Al.xAlrTankCloseToEmpty;
HoldingRegister[1052].1:=gInks[5].Al.xAlrTankCloseToEmpty;
HoldingRegister[1052].2:=gInks[6].Al.xAlrTankCloseToEmpty;
HoldingRegister[1052].3:=gInks[7].Al.xAlrTankCloseToEmpty;
HoldingRegister[1052].4:=gInks[8].Al.xAlrTankCloseToEmpty;
HoldingRegister[1052].5:=gInks[9].Al.xAlrTankCloseToEmpty;
HoldingRegister[1052].6:=gInks[10].Al.xAlrTankCloseToEmpty;
HoldingRegister[1052].7:=gInks[11].Al.xAlrTankCloseToEmpty;
HoldingRegister[1052].8:=gInks[12].Al.xAlrTankCloseToEmpty;
HoldingRegister[1052].9:=gInks[1].Al.xAlrTempTankSensor;
HoldingRegister[1052].10:=gInks[2].Al.xAlrTempTankSensor;
HoldingRegister[1052].11:=gInks[3].Al.xAlrTempTankSensor;
HoldingRegister[1052].12:=gInks[4].Al.xAlrTempTankSensor;
HoldingRegister[1052].13:=gInks[5].Al.xAlrTempTankSensor;
HoldingRegister[1052].14:=gInks[6].Al.xAlrTempTankSensor;
HoldingRegister[1052].15:=gInks[7].Al.xAlrTempTankSensor;
HoldingRegister[1053].0:=gInks[8].Al.xAlrTempTankSensor;
HoldingRegister[1053].1:=gInks[9].Al.xAlrTempTankSensor;
HoldingRegister[1053].2:=gInks[10].Al.xAlrTempTankSensor;
HoldingRegister[1053].3:=gInks[11].Al.xAlrTempTankSensor;
HoldingRegister[1053].4:=gInks[12].Al.xAlrTempTankSensor;
HoldingRegister[1053].5:=gBlock[1].Al.xAlrTempPowerSupply;
HoldingRegister[1053].6:=gBlock[2].Al.xAlrTempPowerSupply;
HoldingRegister[1053].7:=gChiller[1].Alarm.xAlrTempSensBrokn;
HoldingRegister[1053].8:=gChiller[1].St.xEnabled;
HoldingRegister[1053].9:=gMachine.Al.Alarm.xAlrThicknSystemNotSelected;
HoldingRegister[1053].10:=gPhotoCells.status.xInstalled;
HoldingRegister[1053].11:=gTime.Status.TimeUpdated;
HoldingRegister[1053].12:=gMachine.Al.Warning.xSAIBypass;
HoldingRegister[1053].13:=gMachine.Al.Warning.xSAIFault;
HoldingRegister[1053].14:=gMachine.Al.Warning.xSAILowBat;
HoldingRegister[1053].15:=gMachine.Al.Alarm.xAlarmSAIPowerFault;
HoldingRegister[1054].1:=gTransVacuum[1].Status.xInstalled;
HoldingRegister[1054].2:=gTransVacuum[1].Alarms.xAlrBlowersAnyCB;
HoldingRegister[1054].3:=gBlock[1].Al.xAlrEmptyWaterTank;
HoldingRegister[1054].4:=gBlock[2].Al.xAlrEmptyWaterTank;
HoldingRegister[1054].5:=gMachine.Al.Alarm.xAlrDingWrongPosition;
HoldingRegister[1054].6:=gMachine.Al.Alarm.xAlrWrongPhysConf;
HoldingRegister[1054].7:=gBlock[1].Al.xAlrWtrPresSensBroken;
HoldingRegister[1054].8:=gBlock[2].Al.xAlrWtrPresSensBroken;
HoldingRegister[1054].9:=gMachine.Pt.Hw.xSuctionModeAllowed;
HoldingRegister[1055]:=REAL_TO_INT(gBlock[1].Status.rMotorPosition*10);
HoldingRegister[1056]:=REAL_TO_INT(gBlock[2].Status.rMotorPosition*10);
HoldingRegister[1057]:=REAL_TO_INT(gDing.State.rCurrentThicknessStable*10);
HoldingRegister[1058]:=REAL_TO_INT(gMachine.Pt.CT.rMaxTicknessMedia*10);
HoldingRegister[1059]:=REAL_TO_INT(gBelt.states.rMaxSpeed*10);
HoldingRegister[1060]:=REAL_TO_INT(gBelt.states.rCurrentTorque*1);
HoldingRegister[1061]:=REAL_TO_INT(gBelt.states.rTorquePerc*10);
HoldingRegister[1063]:=gMachine.St.Cleaning.iCleaningState;
HoldingRegister[1064]:=gMachine.St.Cleaning.iPieceCounterBtwCleaningsL1;
HoldingRegister[1065]:=gMachine.St.Cleaning.iPieceCounterBtwCleaningsL1;
HoldingRegister[1066]:=gMachine.St.uiLicenseCounter;
HoldingRegister[1067]:=REAL_TO_INT(gDing.State.rOffsetCalibration*10);
HoldingRegister[1068]:=REAL_TO_INT(gInks[1].status.PosPump.rCurrent*100);
HoldingRegister[1069]:=REAL_TO_INT(gInks[2].status.PosPump.rCurrent*100);
HoldingRegister[1070]:=REAL_TO_INT(gInks[3].status.PosPump.rCurrent*100);
HoldingRegister[1071]:=REAL_TO_INT(gInks[4].status.PosPump.rCurrent*100);
HoldingRegister[1072]:=REAL_TO_INT(gInks[5].status.PosPump.rCurrent*100);
HoldingRegister[1073]:=REAL_TO_INT(gInks[6].status.PosPump.rCurrent*100);
HoldingRegister[1074]:=REAL_TO_INT(gInks[7].status.PosPump.rCurrent*100);
HoldingRegister[1075]:=REAL_TO_INT(gInks[8].status.PosPump.rCurrent*100);
HoldingRegister[1076]:=REAL_TO_INT(gInks[9].status.PosPump.rCurrent*100);
HoldingRegister[1077]:=REAL_TO_INT(gInks[10].status.PosPump.rCurrent*100);
HoldingRegister[1078]:=REAL_TO_INT(gInks[11].status.PosPump.rCurrent*100);
HoldingRegister[1079]:=REAL_TO_INT(gInks[12].status.PosPump.rCurrent*100);
HoldingRegister[1080]:=REAL_TO_INT(gInks[1].status.NegPump.rCurrent*100);
HoldingRegister[1081]:=REAL_TO_INT(gInks[2].status.NegPump.rCurrent*100);
HoldingRegister[1082]:=REAL_TO_INT(gInks[3].status.NegPump.rCurrent*100);
HoldingRegister[1083]:=REAL_TO_INT(gInks[4].status.NegPump.rCurrent*100);
HoldingRegister[1084]:=REAL_TO_INT(gInks[5].status.NegPump.rCurrent*100);
HoldingRegister[1085]:=REAL_TO_INT(gInks[6].status.NegPump.rCurrent*100);
HoldingRegister[1086]:=REAL_TO_INT(gInks[7].status.NegPump.rCurrent*100);
HoldingRegister[1087]:=REAL_TO_INT(gInks[8].status.NegPump.rCurrent*100);
HoldingRegister[1088]:=REAL_TO_INT(gInks[9].status.NegPump.rCurrent*100);
HoldingRegister[1089]:=REAL_TO_INT(gInks[10].status.NegPump.rCurrent*100);
HoldingRegister[1090]:=REAL_TO_INT(gInks[11].status.NegPump.rCurrent*100);
HoldingRegister[1091]:=REAL_TO_INT(gInks[12].status.NegPump.rCurrent*100);
HoldingRegister[1092]:=REAL_TO_INT(gInks[1].status.PosPump.rDutyCycleFilling*10);
HoldingRegister[1093]:=REAL_TO_INT(gInks[2].status.PosPump.rDutyCycleFilling*10);
HoldingRegister[1094]:=REAL_TO_INT(gInks[3].status.PosPump.rDutyCycleFilling*10);
HoldingRegister[1095]:=REAL_TO_INT(gInks[4].status.PosPump.rDutyCycleFilling*10);
HoldingRegister[1096]:=REAL_TO_INT(gInks[5].status.PosPump.rDutyCycleFilling*10);
HoldingRegister[1097]:=REAL_TO_INT(gInks[6].status.PosPump.rDutyCycleFilling*10);
HoldingRegister[1098]:=REAL_TO_INT(gInks[7].status.PosPump.rDutyCycleFilling*10);
HoldingRegister[1099]:=REAL_TO_INT(gInks[8].status.PosPump.rDutyCycleFilling*10);
HoldingRegister[1100]:=REAL_TO_INT(gInks[9].status.PosPump.rDutyCycleFilling*10);
HoldingRegister[1101]:=REAL_TO_INT(gInks[10].status.PosPump.rDutyCycleFilling*10);
HoldingRegister[1102]:=REAL_TO_INT(gInks[11].status.PosPump.rDutyCycleFilling*10);
HoldingRegister[1103]:=REAL_TO_INT(gInks[12].status.PosPump.rDutyCycleFilling*10);
HoldingRegister[1104]:=REAL_TO_INT(gInks[1].status.NegPump.rDutyCycleNegative*10);
HoldingRegister[1105]:=REAL_TO_INT(gInks[2].status.NegPump.rDutyCycleNegative*10);
HoldingRegister[1106]:=REAL_TO_INT(gInks[3].status.NegPump.rDutyCycleNegative*10);
HoldingRegister[1107]:=REAL_TO_INT(gInks[4].status.NegPump.rDutyCycleNegative*10);
HoldingRegister[1108]:=REAL_TO_INT(gInks[5].status.NegPump.rDutyCycleNegative*10);
HoldingRegister[1109]:=REAL_TO_INT(gInks[6].status.NegPump.rDutyCycleNegative*10);
HoldingRegister[1110]:=REAL_TO_INT(gInks[7].status.NegPump.rDutyCycleNegative*10);
HoldingRegister[1111]:=REAL_TO_INT(gInks[8].status.NegPump.rDutyCycleNegative*10);
HoldingRegister[1112]:=REAL_TO_INT(gInks[9].status.NegPump.rDutyCycleNegative*10);
HoldingRegister[1113]:=REAL_TO_INT(gInks[10].status.NegPump.rDutyCycleNegative*10);
HoldingRegister[1114]:=REAL_TO_INT(gInks[11].status.NegPump.rDutyCycleNegative*10);
HoldingRegister[1115]:=REAL_TO_INT(gInks[12].status.NegPump.rDutyCycleNegative*10);
HoldingRegister[1116]:=REAL_TO_INT(gInks[1].status.Temp.rDutyCycleTempPowerRed*10);
HoldingRegister[1117]:=REAL_TO_INT(gInks[2].status.Temp.rDutyCycleTempPowerRed*10);
HoldingRegister[1118]:=REAL_TO_INT(gInks[3].status.Temp.rDutyCycleTempPowerRed*10);
HoldingRegister[1119]:=REAL_TO_INT(gInks[4].status.Temp.rDutyCycleTempPowerRed*10);
HoldingRegister[1120]:=REAL_TO_INT(gInks[5].status.Temp.rDutyCycleTempPowerRed*10);
HoldingRegister[1121]:=REAL_TO_INT(gInks[6].status.Temp.rDutyCycleTempPowerRed*10);
HoldingRegister[1122]:=REAL_TO_INT(gInks[7].status.Temp.rDutyCycleTempPowerRed*10);
HoldingRegister[1123]:=REAL_TO_INT(gInks[8].status.Temp.rDutyCycleTempPowerRed*10);
HoldingRegister[1124]:=REAL_TO_INT(gInks[9].status.Temp.rDutyCycleTempPowerRed*10);
HoldingRegister[1125]:=REAL_TO_INT(gInks[10].status.Temp.rDutyCycleTempPowerRed*10);
HoldingRegister[1126]:=REAL_TO_INT(gInks[11].status.Temp.rDutyCycleTempPowerRed*10);
HoldingRegister[1127]:=REAL_TO_INT(gInks[12].status.Temp.rDutyCycleTempPowerRed*10);
HoldingRegister[1128]:=REAL_TO_INT(gInks[1].status.Temp.rDutyCycleTempPowerRedTank*10);
HoldingRegister[1129]:=REAL_TO_INT(gInks[2].status.Temp.rDutyCycleTempPowerRedTank*10);
HoldingRegister[1130]:=REAL_TO_INT(gInks[3].status.Temp.rDutyCycleTempPowerRedTank*10);
HoldingRegister[1131]:=REAL_TO_INT(gInks[4].status.Temp.rDutyCycleTempPowerRedTank*10);
HoldingRegister[1132]:=REAL_TO_INT(gInks[5].status.Temp.rDutyCycleTempPowerRedTank*10);
HoldingRegister[1133]:=REAL_TO_INT(gInks[6].status.Temp.rDutyCycleTempPowerRedTank*10);
HoldingRegister[1134]:=REAL_TO_INT(gInks[7].status.Temp.rDutyCycleTempPowerRedTank*10);
HoldingRegister[1135]:=REAL_TO_INT(gInks[8].status.Temp.rDutyCycleTempPowerRedTank*10);
HoldingRegister[1136]:=REAL_TO_INT(gInks[9].status.Temp.rDutyCycleTempPowerRedTank*10);
HoldingRegister[1137]:=REAL_TO_INT(gInks[10].status.Temp.rDutyCycleTempPowerRedTank*10);
HoldingRegister[1138]:=REAL_TO_INT(gInks[11].status.Temp.rDutyCycleTempPowerRedTank*10);
HoldingRegister[1139]:=REAL_TO_INT(gInks[12].status.Temp.rDutyCycleTempPowerRedTank*10);
HoldingRegister[1140]:=gBlock[1].Status.iBlockState;
HoldingRegister[1141]:=gBlock[2].Status.iBlockState;
HoldingRegister[1142]:=gMachine.St.iAutoModeSW;
HoldingRegister[1143]:=gMachine.St.iFaultRunPlc;
HoldingRegister[1144]:=REAL_TO_INT(gTransVacuum[1].Status.Blower.rDutyCycle*10);
HoldingRegister[1145]:=gInks[1].status.iInkStateSw;
HoldingRegister[1146]:=gInks[2].status.iInkStateSw;
HoldingRegister[1147]:=gInks[3].status.iInkStateSw;
HoldingRegister[1148]:=gInks[4].status.iInkStateSw;
HoldingRegister[1149]:=gInks[5].status.iInkStateSw;
HoldingRegister[1150]:=gInks[6].status.iInkStateSw;
HoldingRegister[1151]:=gInks[7].status.iInkStateSw;
HoldingRegister[1152]:=gInks[8].status.iInkStateSw;
HoldingRegister[1153]:=gInks[9].status.iInkStateSw;
HoldingRegister[1154]:=gInks[10].status.iInkStateSw;
HoldingRegister[1155]:=gInks[11].status.iInkStateSw;
HoldingRegister[1156]:=gInks[12].status.iInkStateSw;
HoldingRegister[1158]:=gBlock[1].Status.Icla.iIntensityCleanMotor;
HoldingRegister[1159]:=gBlock[2].Status.Icla.iIntensityCleanMotor;
HoldingRegister[1160]:=gBlock[1].Status.Motor.iIntensityVertMotor;
HoldingRegister[1161]:=gBlock[2].Status.Motor.iIntensityVertMotor;
HoldingRegister[1162]:=gInks[1].status.Tank.iDipositLevel;
HoldingRegister[1163]:=gInks[2].status.Tank.iDipositLevel;
HoldingRegister[1164]:=gInks[3].status.Tank.iDipositLevel;
HoldingRegister[1165]:=gInks[4].status.Tank.iDipositLevel;
HoldingRegister[1166]:=gInks[5].status.Tank.iDipositLevel;
HoldingRegister[1167]:=gInks[6].status.Tank.iDipositLevel;
HoldingRegister[1168]:=gInks[7].status.Tank.iDipositLevel;
HoldingRegister[1169]:=gInks[8].status.Tank.iDipositLevel;
HoldingRegister[1170]:=gInks[9].status.Tank.iDipositLevel;
HoldingRegister[1171]:=gInks[10].status.Tank.iDipositLevel;
HoldingRegister[1172]:=gInks[11].status.Tank.iDipositLevel;
HoldingRegister[1173]:=gInks[12].status.Tank.iDipositLevel;
HoldingRegister[1174]:=gInks[1].status.Tank.iStatusTankDigital;
HoldingRegister[1175]:=gInks[2].status.Tank.iStatusTankDigital;
HoldingRegister[1176]:=gInks[3].status.Tank.iStatusTankDigital;
HoldingRegister[1177]:=gInks[4].status.Tank.iStatusTankDigital;
HoldingRegister[1178]:=gInks[5].status.Tank.iStatusTankDigital;
HoldingRegister[1179]:=gInks[6].status.Tank.iStatusTankDigital;
HoldingRegister[1180]:=gInks[7].status.Tank.iStatusTankDigital;
HoldingRegister[1181]:=gInks[8].status.Tank.iStatusTankDigital;
HoldingRegister[1182]:=gInks[9].status.Tank.iStatusTankDigital;
HoldingRegister[1183]:=gInks[10].status.Tank.iStatusTankDigital;
HoldingRegister[1184]:=gInks[11].status.Tank.iStatusTankDigital;
HoldingRegister[1185]:=gInks[12].status.Tank.iStatusTankDigital;
HoldingRegister[1186]:=gMachine.Lg.iTilesCounterToClean;
HoldingRegister[1187]:=gMachine.Lg.iTilesCounterToCleanBeltTop;
HoldingRegister[1188]:=REAL_TO_INT(gInks[1].parSw.NegPump.rLowerLimMeniscusCritical*10);
HoldingRegister[1189]:=REAL_TO_INT(gInks[2].parSw.NegPump.rLowerLimMeniscusCritical*10);
HoldingRegister[1190]:=REAL_TO_INT(gInks[3].parSw.NegPump.rLowerLimMeniscusCritical*10);
HoldingRegister[1191]:=REAL_TO_INT(gInks[4].parSw.NegPump.rLowerLimMeniscusCritical*10);
HoldingRegister[1192]:=REAL_TO_INT(gInks[5].parSw.NegPump.rLowerLimMeniscusCritical*10);
HoldingRegister[1193]:=REAL_TO_INT(gInks[6].parSw.NegPump.rLowerLimMeniscusCritical*10);
HoldingRegister[1194]:=REAL_TO_INT(gInks[7].parSw.NegPump.rLowerLimMeniscusCritical*10);
HoldingRegister[1195]:=REAL_TO_INT(gInks[8].parSw.NegPump.rLowerLimMeniscusCritical*10);
HoldingRegister[1196]:=REAL_TO_INT(gInks[9].parSw.NegPump.rLowerLimMeniscusCritical*10);
HoldingRegister[1197]:=REAL_TO_INT(gInks[10].parSw.NegPump.rLowerLimMeniscusCritical*10);
HoldingRegister[1198]:=REAL_TO_INT(gInks[11].parSw.NegPump.rLowerLimMeniscusCritical*10);
HoldingRegister[1199]:=REAL_TO_INT(gInks[12].parSw.NegPump.rLowerLimMeniscusCritical*10);
HoldingRegister[1200]:=REAL_TO_INT(gInks[1].status.rMeniscus*10);
HoldingRegister[1201]:=REAL_TO_INT(gInks[2].status.rMeniscus*10);
HoldingRegister[1202]:=REAL_TO_INT(gInks[3].status.rMeniscus*10);
HoldingRegister[1203]:=REAL_TO_INT(gInks[4].status.rMeniscus*10);
HoldingRegister[1204]:=REAL_TO_INT(gInks[5].status.rMeniscus*10);
HoldingRegister[1205]:=REAL_TO_INT(gInks[6].status.rMeniscus*10);
HoldingRegister[1206]:=REAL_TO_INT(gInks[7].status.rMeniscus*10);
HoldingRegister[1207]:=REAL_TO_INT(gInks[8].status.rMeniscus*10);
HoldingRegister[1208]:=REAL_TO_INT(gInks[9].status.rMeniscus*10);
HoldingRegister[1209]:=REAL_TO_INT(gInks[10].status.rMeniscus*10);
HoldingRegister[1210]:=REAL_TO_INT(gInks[11].status.rMeniscus*10);
HoldingRegister[1211]:=REAL_TO_INT(gInks[12].status.rMeniscus*10);
HoldingRegister[1215]:=gMachine.St.iMachineModelCodeSW;
HoldingRegister[1216]:=gBlock[1].Status.Motor.ErrorID;
HoldingRegister[1217]:=gBlock[2].Status.Motor.ErrorID;
HoldingRegister[1218]:=gBelt.states.ErrorId;
HoldingRegister[1219]:=gBlock[1].Status.Icla.ErrorNumber;
HoldingRegister[1220]:=gBlock[2].Status.Icla.ErrorNumber;
HoldingRegister[1221]:=REAL_TO_INT(gBlock[1].parameters.Motor.rMaxCleanOffsetTech*10);
HoldingRegister[1222]:=REAL_TO_INT(gBlock[2].parameters.Motor.rMaxCleanOffsetTech*10);
HoldingRegister[1223]:=REAL_TO_INT(gBlock[1].parameters.Motor.rMinCleanOffsetTech*10);
HoldingRegister[1224]:=REAL_TO_INT(gBlock[2].parameters.Motor.rMinCleanOffsetTech*10);
HoldingRegister[1249]:=gBlock[1].Status.Motor.iActTorque;
HoldingRegister[1250]:=gBlock[2].Status.Motor.iActTorque;
HoldingRegister[1251]:=REAL_TO_INT(gPhotoCells.status.rPositionMotor*10);
HoldingRegister[1252]:=REAL_TO_INT(gBlock[1].Status.Icla.rCurrentPosition*1);
HoldingRegister[1253]:=REAL_TO_INT(gBlock[2].Status.Icla.rCurrentPosition*1);
HoldingRegister[1254]:=REAL_TO_INT(gMachine.Pt.rMaxPrintHeadPos*1);
HoldingRegister[1255]:=REAL_TO_INT(gMachine.Pt.rMinPrintHeadPos*1);
HoldingRegister[1256]:=gMachine.In.iRelieve1;
HoldingRegister[1257]:=gMachine.In.iRelieve2;
HoldingRegister[1258]:=gBlock[1].Status.Icla.iSpeed;
HoldingRegister[1259]:=gBlock[2].Status.Icla.iSpeed;
HoldingRegister[1260]:=gMachine.Lg.iDiffPiecesStrobeProductDetect;
HoldingRegister[1261]:=REAL_TO_INT(gInks[1].status.Temp.rTemp*10);
HoldingRegister[1262]:=REAL_TO_INT(gInks[2].status.Temp.rTemp*10);
HoldingRegister[1263]:=REAL_TO_INT(gInks[3].status.Temp.rTemp*10);
HoldingRegister[1264]:=REAL_TO_INT(gInks[4].status.Temp.rTemp*10);
HoldingRegister[1265]:=REAL_TO_INT(gInks[5].status.Temp.rTemp*10);
HoldingRegister[1266]:=REAL_TO_INT(gInks[6].status.Temp.rTemp*10);
HoldingRegister[1267]:=REAL_TO_INT(gInks[7].status.Temp.rTemp*10);
HoldingRegister[1268]:=REAL_TO_INT(gInks[8].status.Temp.rTemp*10);
HoldingRegister[1269]:=REAL_TO_INT(gInks[9].status.Temp.rTemp*10);
HoldingRegister[1270]:=REAL_TO_INT(gInks[10].status.Temp.rTemp*10);
HoldingRegister[1271]:=REAL_TO_INT(gInks[11].status.Temp.rTemp*10);
HoldingRegister[1272]:=REAL_TO_INT(gInks[12].status.Temp.rTemp*10);
HoldingRegister[1273]:=REAL_TO_INT(gInks[1].status.Temp.rTempTank*10);
HoldingRegister[1274]:=REAL_TO_INT(gInks[2].status.Temp.rTempTank*10);
HoldingRegister[1275]:=REAL_TO_INT(gInks[3].status.Temp.rTempTank*10);
HoldingRegister[1276]:=REAL_TO_INT(gInks[4].status.Temp.rTempTank*10);
HoldingRegister[1277]:=REAL_TO_INT(gInks[5].status.Temp.rTempTank*10);
HoldingRegister[1278]:=REAL_TO_INT(gInks[6].status.Temp.rTempTank*10);
HoldingRegister[1279]:=REAL_TO_INT(gInks[7].status.Temp.rTempTank*10);
HoldingRegister[1280]:=REAL_TO_INT(gInks[8].status.Temp.rTempTank*10);
HoldingRegister[1281]:=REAL_TO_INT(gInks[9].status.Temp.rTempTank*10);
HoldingRegister[1282]:=REAL_TO_INT(gInks[10].status.Temp.rTempTank*10);
HoldingRegister[1283]:=REAL_TO_INT(gInks[11].status.Temp.rTempTank*10);
HoldingRegister[1284]:=REAL_TO_INT(gInks[12].status.Temp.rTempTank*10);
HoldingRegister[1285]:=TIME_TO_SECONDS_COMS(gInksConstants.tiDripTimeMax)/1;
HoldingRegister[1286]:=TIME_TO_SECONDS_COMS(gInksConstants.tiDripTimeMin)/1;
HoldingRegister[1287]:=gTime.Status.SwState;
HoldingRegister[1288]:=TIME_TO_MILLISECONDS_COMS(gInks[1].status.tiInReverseManual)*100;
HoldingRegister[1289]:=TIME_TO_MILLISECONDS_COMS(gInks[2].status.tiInReverseManual)*100;
HoldingRegister[1290]:=TIME_TO_MILLISECONDS_COMS(gInks[3].status.tiInReverseManual)*100;
HoldingRegister[1291]:=TIME_TO_MILLISECONDS_COMS(gInks[4].status.tiInReverseManual)*100;
HoldingRegister[1292]:=TIME_TO_MILLISECONDS_COMS(gInks[5].status.tiInReverseManual)*100;
HoldingRegister[1293]:=TIME_TO_MILLISECONDS_COMS(gInks[6].status.tiInReverseManual)*100;
HoldingRegister[1294]:=TIME_TO_MILLISECONDS_COMS(gInks[7].status.tiInReverseManual)*100;
HoldingRegister[1295]:=TIME_TO_MILLISECONDS_COMS(gInks[8].status.tiInReverseManual)*100;
HoldingRegister[1296]:=TIME_TO_MILLISECONDS_COMS(gInks[9].status.tiInReverseManual)*100;
HoldingRegister[1297]:=TIME_TO_MILLISECONDS_COMS(gInks[10].status.tiInReverseManual)*100;
HoldingRegister[1298]:=TIME_TO_MILLISECONDS_COMS(gInks[11].status.tiInReverseManual)*100;
HoldingRegister[1299]:=TIME_TO_MILLISECONDS_COMS(gInks[12].status.tiInReverseManual)*100;
HoldingRegister[1300]:=REAL_TO_INT(gInks[1].parSw.NegPump.rUpperLimMeniscusCritical*10);
HoldingRegister[1301]:=REAL_TO_INT(gInks[2].parSw.NegPump.rUpperLimMeniscusCritical*10);
HoldingRegister[1302]:=REAL_TO_INT(gInks[3].parSw.NegPump.rUpperLimMeniscusCritical*10);
HoldingRegister[1303]:=REAL_TO_INT(gInks[4].parSw.NegPump.rUpperLimMeniscusCritical*10);
HoldingRegister[1304]:=REAL_TO_INT(gInks[5].parSw.NegPump.rUpperLimMeniscusCritical*10);
HoldingRegister[1305]:=REAL_TO_INT(gInks[6].parSw.NegPump.rUpperLimMeniscusCritical*10);
HoldingRegister[1306]:=REAL_TO_INT(gInks[7].parSw.NegPump.rUpperLimMeniscusCritical*10);
HoldingRegister[1307]:=REAL_TO_INT(gInks[8].parSw.NegPump.rUpperLimMeniscusCritical*10);
HoldingRegister[1308]:=REAL_TO_INT(gInks[9].parSw.NegPump.rUpperLimMeniscusCritical*10);
HoldingRegister[1309]:=REAL_TO_INT(gInks[10].parSw.NegPump.rUpperLimMeniscusCritical*10);
HoldingRegister[1310]:=REAL_TO_INT(gInks[11].parSw.NegPump.rUpperLimMeniscusCritical*10);
HoldingRegister[1311]:=REAL_TO_INT(gInks[12].parSw.NegPump.rUpperLimMeniscusCritical*10);
HoldingRegister[1312]:=REAL_TO_INT(gInks[1].status.rVacuum1*10);
HoldingRegister[1313]:=REAL_TO_INT(gInks[2].status.rVacuum1*10);
HoldingRegister[1314]:=REAL_TO_INT(gInks[3].status.rVacuum1*10);
HoldingRegister[1315]:=REAL_TO_INT(gInks[4].status.rVacuum1*10);
HoldingRegister[1316]:=REAL_TO_INT(gInks[5].status.rVacuum1*10);
HoldingRegister[1317]:=REAL_TO_INT(gInks[6].status.rVacuum1*10);
HoldingRegister[1318]:=REAL_TO_INT(gInks[7].status.rVacuum1*10);
HoldingRegister[1319]:=REAL_TO_INT(gInks[8].status.rVacuum1*10);
HoldingRegister[1320]:=REAL_TO_INT(gInks[9].status.rVacuum1*10);
HoldingRegister[1321]:=REAL_TO_INT(gInks[10].status.rVacuum1*10);
HoldingRegister[1322]:=REAL_TO_INT(gInks[11].status.rVacuum1*10);
HoldingRegister[1323]:=REAL_TO_INT(gInks[12].status.rVacuum1*10);
HoldingRegister[1324]:=REAL_TO_INT(gInks[1].status.rVacuum2*10);
HoldingRegister[1325]:=REAL_TO_INT(gInks[2].status.rVacuum2*10);
HoldingRegister[1326]:=REAL_TO_INT(gInks[3].status.rVacuum2*10);
HoldingRegister[1327]:=REAL_TO_INT(gInks[4].status.rVacuum2*10);
HoldingRegister[1328]:=REAL_TO_INT(gInks[5].status.rVacuum2*10);
HoldingRegister[1329]:=REAL_TO_INT(gInks[6].status.rVacuum2*10);
HoldingRegister[1330]:=REAL_TO_INT(gInks[7].status.rVacuum2*10);
HoldingRegister[1331]:=REAL_TO_INT(gInks[8].status.rVacuum2*10);
HoldingRegister[1332]:=REAL_TO_INT(gInks[9].status.rVacuum2*10);
HoldingRegister[1333]:=REAL_TO_INT(gInks[10].status.rVacuum2*10);
HoldingRegister[1334]:=REAL_TO_INT(gInks[11].status.rVacuum2*10);
HoldingRegister[1335]:=REAL_TO_INT(gInks[12].status.rVacuum2*10);
HoldingRegister[1336]:=REAL_TO_INT(gTransVacuum[1].Parameters.Hw.rAreaWidth*1);
HoldingRegister[1337]:=REAL_TO_INT(gTransVacuum[1].Parameters.Hw.rCentralAreaWithoutVacuum*1);
HoldingRegister[1338]:=REAL_TO_INT(gTransVacuum[1].Status.rPressurePerc*10);
HoldingRegister[1339]:=gTransVacuum[1].Parameters.Hw.iTotalAreas;
HoldingRegister[1340]:=gPLC.iVarsVersion3;
HoldingRegister[1341]:=gBlock[1].parameters.Icla.iMaxSpeedCleanMotorFwd;
HoldingRegister[1342]:=gBlock[1].parameters.Icla.iMinSpeedCleanMotorFwd;
HoldingRegister[1343]:=REAL_TO_INT(gBelt.states.rCurrentSpeed*10);
UDINTToComms(gMachine.Lg.udiPiecesCounterL1,1344,ADR(HoldingRegister));
UDINTToComms(gMachine.Lg.udiPiecesCounterL2,1346,ADR(HoldingRegister));
UDINTToComms(gMachine.Lg.udiDifCounters,1348,ADR(HoldingRegister));
UDINTToComms(gBelt.Log.udiKmBand,1350,ADR(HoldingRegister));
UDINTToComms(gMachine.St.Cleaning.MinutesInProdForClean,1352,ADR(HoldingRegister));
UDINTToComms(gMachine.St.Cleaning.MinutesInStopForClean,1354,ADR(HoldingRegister));
UDINTToComms(gMachine.Lg.udiTileCounterBalluffLaser,1356,ADR(HoldingRegister));
UDINTToComms(gMachine.Lg.udiTileCounterTriggerLaser,1358,ADR(HoldingRegister));
HoldingRegister[3000]:=TIME_TO_SECONDS_COMS(gMachine.parSw.Clean.tiBetweenCleaningBlocks)/1;
HoldingRegister[3001]:=gMachine.parSw.Clean.iCleaningType;
HoldingRegister[3002]:=REAL_TO_INT(gDing.parSw.rCalibrationValue*10);
HoldingRegister[3003]:=REAL_TO_INT(gMachine.parSw.Media.rThickness*10);
HoldingRegister[3004]:=REAL_TO_INT(gInks[1].parSw.NegPump.rLimitMeniscusDiffWarning*10);
HoldingRegister[3005]:=REAL_TO_INT(gInks[2].parSw.NegPump.rLimitMeniscusDiffWarning*10);
HoldingRegister[3006]:=REAL_TO_INT(gInks[3].parSw.NegPump.rLimitMeniscusDiffWarning*10);
HoldingRegister[3007]:=REAL_TO_INT(gInks[4].parSw.NegPump.rLimitMeniscusDiffWarning*10);
HoldingRegister[3008]:=REAL_TO_INT(gInks[5].parSw.NegPump.rLimitMeniscusDiffWarning*10);
HoldingRegister[3009]:=REAL_TO_INT(gInks[6].parSw.NegPump.rLimitMeniscusDiffWarning*10);
HoldingRegister[3010]:=REAL_TO_INT(gInks[7].parSw.NegPump.rLimitMeniscusDiffWarning*10);
HoldingRegister[3011]:=REAL_TO_INT(gInks[8].parSw.NegPump.rLimitMeniscusDiffWarning*10);
HoldingRegister[3012]:=REAL_TO_INT(gInks[9].parSw.NegPump.rLimitMeniscusDiffWarning*10);
HoldingRegister[3013]:=REAL_TO_INT(gInks[10].parSw.NegPump.rLimitMeniscusDiffWarning*10);
HoldingRegister[3014]:=REAL_TO_INT(gInks[11].parSw.NegPump.rLimitMeniscusDiffWarning*10);
HoldingRegister[3015]:=REAL_TO_INT(gInks[12].parSw.NegPump.rLimitMeniscusDiffWarning*10);
HoldingRegister[3016]:=REAL_TO_INT(gMachine.parSw.rMarginPrint*10);
HoldingRegister[3017]:=REAL_TO_INT(gMachine.parSw.Media.rWidth*10);
HoldingRegister[3018]:=REAL_TO_INT(gNonCrash[1].parSw.rGearBox*1);
HoldingRegister[3019]:=REAL_TO_INT(gNonCrash[1].parSw.rPerimeter*10);
HoldingRegister[3020]:=REAL_TO_INT(gNonCrash[1].parSw.rSpeedOffset*10);
HoldingRegister[3021]:=REAL_TO_INT(gMachine.parSw.rFirstHeadPosition*1);
HoldingRegister[3022]:=REAL_TO_INT(gMachine.parSw.rLastHeadPosition*1);
HoldingRegister[3023]:=REAL_TO_INT(gInks[1].parSw.PosPump.rSetPoint*10);
HoldingRegister[3024]:=REAL_TO_INT(gInks[2].parSw.PosPump.rSetPoint*10);
HoldingRegister[3025]:=REAL_TO_INT(gInks[3].parSw.PosPump.rSetPoint*10);
HoldingRegister[3026]:=REAL_TO_INT(gInks[4].parSw.PosPump.rSetPoint*10);
HoldingRegister[3027]:=REAL_TO_INT(gInks[5].parSw.PosPump.rSetPoint*10);
HoldingRegister[3028]:=REAL_TO_INT(gInks[6].parSw.PosPump.rSetPoint*10);
HoldingRegister[3029]:=REAL_TO_INT(gInks[7].parSw.PosPump.rSetPoint*10);
HoldingRegister[3030]:=REAL_TO_INT(gInks[8].parSw.PosPump.rSetPoint*10);
HoldingRegister[3031]:=REAL_TO_INT(gInks[9].parSw.PosPump.rSetPoint*10);
HoldingRegister[3032]:=REAL_TO_INT(gInks[10].parSw.PosPump.rSetPoint*10);
HoldingRegister[3033]:=REAL_TO_INT(gInks[11].parSw.PosPump.rSetPoint*10);
HoldingRegister[3034]:=REAL_TO_INT(gInks[12].parSw.PosPump.rSetPoint*10);
HoldingRegister[3035]:=REAL_TO_INT(gInks[1].parSw.NegPump.rSetPointMeniscus*1);
HoldingRegister[3036]:=REAL_TO_INT(gInks[2].parSw.NegPump.rSetPointMeniscus*1);
HoldingRegister[3037]:=REAL_TO_INT(gInks[3].parSw.NegPump.rSetPointMeniscus*1);
HoldingRegister[3038]:=REAL_TO_INT(gInks[4].parSw.NegPump.rSetPointMeniscus*1);
HoldingRegister[3039]:=REAL_TO_INT(gInks[5].parSw.NegPump.rSetPointMeniscus*1);
HoldingRegister[3040]:=REAL_TO_INT(gInks[6].parSw.NegPump.rSetPointMeniscus*1);
HoldingRegister[3041]:=REAL_TO_INT(gInks[7].parSw.NegPump.rSetPointMeniscus*1);
HoldingRegister[3042]:=REAL_TO_INT(gInks[8].parSw.NegPump.rSetPointMeniscus*1);
HoldingRegister[3043]:=REAL_TO_INT(gInks[9].parSw.NegPump.rSetPointMeniscus*1);
HoldingRegister[3044]:=REAL_TO_INT(gInks[10].parSw.NegPump.rSetPointMeniscus*1);
HoldingRegister[3045]:=REAL_TO_INT(gInks[11].parSw.NegPump.rSetPointMeniscus*1);
HoldingRegister[3046]:=REAL_TO_INT(gInks[12].parSw.NegPump.rSetPointMeniscus*1);
HoldingRegister[3047]:=REAL_TO_INT(gInks[1].parSw.Temp.rSetPointTemp*10);
HoldingRegister[3048]:=REAL_TO_INT(gInks[2].parSw.Temp.rSetPointTemp*10);
HoldingRegister[3049]:=REAL_TO_INT(gInks[3].parSw.Temp.rSetPointTemp*10);
HoldingRegister[3050]:=REAL_TO_INT(gInks[4].parSw.Temp.rSetPointTemp*10);
HoldingRegister[3051]:=REAL_TO_INT(gInks[5].parSw.Temp.rSetPointTemp*10);
HoldingRegister[3052]:=REAL_TO_INT(gInks[6].parSw.Temp.rSetPointTemp*10);
HoldingRegister[3053]:=REAL_TO_INT(gInks[7].parSw.Temp.rSetPointTemp*10);
HoldingRegister[3054]:=REAL_TO_INT(gInks[8].parSw.Temp.rSetPointTemp*10);
HoldingRegister[3055]:=REAL_TO_INT(gInks[9].parSw.Temp.rSetPointTemp*10);
HoldingRegister[3056]:=REAL_TO_INT(gInks[10].parSw.Temp.rSetPointTemp*10);
HoldingRegister[3057]:=REAL_TO_INT(gInks[11].parSw.Temp.rSetPointTemp*10);
HoldingRegister[3058]:=REAL_TO_INT(gInks[12].parSw.Temp.rSetPointTemp*10);
HoldingRegister[3071]:=REAL_TO_INT(gMachine.parSw.rBeltSpeedSetPoint*10);
HoldingRegister[3072]:=REAL_TO_INT(gInks[1].parSw.NegPump.rSetPointManual*10);
HoldingRegister[3073]:=REAL_TO_INT(gInks[2].parSw.NegPump.rSetPointManual*10);
HoldingRegister[3074]:=REAL_TO_INT(gInks[3].parSw.NegPump.rSetPointManual*10);
HoldingRegister[3075]:=REAL_TO_INT(gInks[4].parSw.NegPump.rSetPointManual*10);
HoldingRegister[3076]:=REAL_TO_INT(gInks[5].parSw.NegPump.rSetPointManual*10);
HoldingRegister[3077]:=REAL_TO_INT(gInks[6].parSw.NegPump.rSetPointManual*10);
HoldingRegister[3078]:=REAL_TO_INT(gInks[7].parSw.NegPump.rSetPointManual*10);
HoldingRegister[3079]:=REAL_TO_INT(gInks[8].parSw.NegPump.rSetPointManual*10);
HoldingRegister[3080]:=REAL_TO_INT(gInks[9].parSw.NegPump.rSetPointManual*10);
HoldingRegister[3081]:=REAL_TO_INT(gInks[10].parSw.NegPump.rSetPointManual*10);
HoldingRegister[3082]:=REAL_TO_INT(gInks[11].parSw.NegPump.rSetPointManual*10);
HoldingRegister[3083]:=REAL_TO_INT(gInks[12].parSw.NegPump.rSetPointManual*10);
HoldingRegister[3084]:=REAL_TO_INT(gInks[1].parSw.PosPump.rSetPointManual*1);
HoldingRegister[3085]:=REAL_TO_INT(gInks[2].parSw.PosPump.rSetPointManual*1);
HoldingRegister[3086]:=REAL_TO_INT(gInks[3].parSw.PosPump.rSetPointManual*1);
HoldingRegister[3087]:=REAL_TO_INT(gInks[4].parSw.PosPump.rSetPointManual*1);
HoldingRegister[3088]:=REAL_TO_INT(gInks[5].parSw.PosPump.rSetPointManual*1);
HoldingRegister[3089]:=REAL_TO_INT(gInks[6].parSw.PosPump.rSetPointManual*1);
HoldingRegister[3090]:=REAL_TO_INT(gInks[7].parSw.PosPump.rSetPointManual*1);
HoldingRegister[3091]:=REAL_TO_INT(gInks[8].parSw.PosPump.rSetPointManual*1);
HoldingRegister[3092]:=REAL_TO_INT(gInks[9].parSw.PosPump.rSetPointManual*1);
HoldingRegister[3093]:=REAL_TO_INT(gInks[10].parSw.PosPump.rSetPointManual*1);
HoldingRegister[3094]:=REAL_TO_INT(gInks[11].parSw.PosPump.rSetPointManual*1);
HoldingRegister[3095]:=REAL_TO_INT(gInks[12].parSw.PosPump.rSetPointManual*1);
HoldingRegister[3096]:=TIME_TO_SECONDS_COMS(gMachine.parSw.tiDelayConsent)/1;
HoldingRegister[3097]:=REAL_TO_INT(gPhotoCells.parSw.rThicknessReference*10);
HoldingRegister[3098]:=TIME_TO_MINUTES(gMachine.parSw.Clean.tiToCleanWhenPrinterStopped)/1;
HoldingRegister[3099]:=gTime.Params.UTCTimeZone;
HoldingRegister[3100]:=gMachine.parSw.Clean.iCleanMotorSpeedFwd;
HoldingRegister[3101]:=gMachine.parSw.Clean.iCleanMotorSpeedBwd;
END_ACTION
```

#### Alarms.st
```iecst
ACTION AlarmKernelPLCComms:

	//Current implementation. Like this to avoid the "not used" messages during compiling
	IF FALSE THEN
		AlarmKernelPLCCommsSocket;
	END_IF

END_ACTION

ACTION AlarmKernelPLCCommsSocket:

	//status_adr := PV_xgetadr(ADR('FB_BRSE_MBT_Server'), ADR(pv_adr), ADR(data_len));(* get the address and the length of PV *)

	status_adr := PV_xgetadr(ADR(nameVar), ADR(pv_adr), ADR(data_len));(* get the address and the length of PV *)
	memcpy(ADR(theValue), pv_adr, data_len);

	iClientsConnected := 0;
	FOR iClient:=0 TO BRSE_MBT_MAX_CLIENT DO
		nameVar := '::FB_BRSE_MBT_Server.Clients[';
		brsitoa(iClient, ADR(strAux));
		strcat(ADR(nameVar), ADR(strAux));
		strcat(ADR(nameVar), ADR('].State'));
		status_adr := PV_xgetadr(ADR(nameVar), ADR(pv_adr), ADR(data_len));(* get the address and the length of PV *)
		memcpy(ADR(theValue), pv_adr, data_len);

		//0=no client, 1=receiving, 2=sending, 9=disconnecting
		IF theValue=2 OR theValue=3 THEN
			iClientsConnected := iClientsConnected + 1;
		END_IF

	END_FOR;

	T_AlarmComPcPlc.IN:= iClientsConnected > 0;
	T_AlarmComPcPlc.PT:= T#10S;	//This is changed to 45secs
	T_AlarmComPcPlc();

	IF EDGEPOS (T_AlarmComPcPlc.Q) THEN
		gMachine.Al.Alarm.xAlarmComPcPLC:= TRUE;
	END_IF;

END_ACTION
```

#### WriteSerialName.st
```iecst
ACTION WriteSerialName:

	strSerialName ACCESS ADR(HoldingRegister[SERIAL_NAME_STATUS_ADR]);
	strSerialName := gMachine.St.HwData.SerialNumber;

END_ACTION
```

#### Variables.var - Local variables
```iecst
VAR
	xStarted : BOOL := FALSE;
	xClenanCommsArray : BOOL;
	iIndexCommsArray : UINT;
	iClient : USINT;
	status_adr : UINT;
	data_len : UDINT;
	nameVar : STRING[180] := '::FB_BRSE_MBT_Server.Clients[0].State';
	pv_adr : UDINT;
	theValue : UINT;
	iClientsConnected : USINT;
	strAux : STRING[10];
	strSerialName : REFERENCE TO STRING[80];
END_VAR
```

### SimMachine.typ
```iecst
TYPE
	SimMachineType :
		(
		SIM_MACHINE_REAL,
		SIM_MACHINE_2B12BAR,
		SIM_MACHINE_1B6BAR,
		SIM_MACHINE_1B2BAR,
		SIM_MACHINE_P5_WAT,
		SIM_MACHINE_P4_CBK,
		SIM_MACHINE_S1400_VAC_PWRLNK,
		SIM_MACHINE_S1400_VAC_CAN,
		SIM_MACHINE_NZ2,
		SIM_MACHINE_NZ2_UV,
		SIM_MACHINE_NZ2_UV_WHITE,
		SIM_MACHINE_CUBE,
		SIM_MACHINE_CUBE_GULLIVER,
		SIM_MACHINE_MECANO_UV_WHITE,
		SIM_MACHINE_MECANO_UV_OPV,
		SIM_MACHINE_MECANO_UV_WHITE_OPV
		);
	SimMachineConsent_typ : 	STRUCT
		xRaiseUpWithNoConsent : BOOL;
	END_STRUCT;
	SimMachineMedia_typ : 	STRUCT
		rMediaThickness : REAL := 15.0; (*Value in mm*)
		xMediaPresent : BOOL; (*To enter one media*)
		xRushProof : BOOL;
		xContinuousMediaPresent : BOOL; (*To constantly entering media in printer*)
		xMediaIfFeederFeeding : BOOL;
	END_STRUCT;
	SimMachineUPSCommand : 	STRUCT
		xRaiseLowBat : BOOL;
		xRaisePowerFault : BOOL;
	END_STRUCT;
	SimMachineLogTest : 	STRUCT
		xCommand : BOOL;
		Text : STRING[80];
	END_STRUCT;
	SimMachineCommand_typ : 	STRUCT
		xToAuto : BOOL; (*Edge command*)
		xToManual : BOOL; (*Edge command*)
		xToZero : BOOL; (*Edge command*)
		xToProduction : BOOL; (*Edge command*)
		Media : SimMachineMedia_typ;
		UPS : SimMachineUPSCommand;
		Consent : SimMachineConsent_typ;
		xStain : BOOL;
		LogTests : SimMachineLogTest;
	END_STRUCT;
	SimMachineSignals_typ : 	STRUCT
		xProductDetectL1 : BOOL; (*Variable to simulate the Product Detect in Simulation*)
		xProductDetectL2 : BOOL; (*Variable to simulate the Product Detect in Simulation*)
		xPDCarriageSignalL1 : BOOL; (*ProductDetect Signal coming from the Carriage Board*)
		xPDCarriageSignalL2 : BOOL; (*ProductDetect Signal coming from the Carriage Board*)
	END_STRUCT;
	SimMachineStackParameters_typ : 	STRUCT
		xLoadNewMedia : BOOL;
		xLoadNewMediaEnergy : BOOL;
		iMediaQuantityToKeepLoaded : USINT;
	END_STRUCT;
	SimMachineParameters_typ : 	STRUCT
		xRunWithKernel : BOOL;
		MachineType : SimMachineType := SIM_MACHINE_REAL;
		DryerType : SimDryerType := SIM_DRYER_NOZ2_NIR;
		xAutoMediaPresent : BOOL;
		Stack : SimMachineStackParameters_typ;
		rStainGap : REAL;
		rStainLength : REAL;
	END_STRUCT;
	SimMachine_typ : 	STRUCT
		Commands : SimMachineCommand_typ;
		Parameters : SimMachineParameters_typ;
		Signals : SimMachineSignals_typ;
	END_STRUCT;
END_TYPE
```

### SimMachineGen.var
```iecst
VAR
	gTraySim : ARRAY[0..MAX_LAST_BLOCK] OF stTraySim;
	gIclaSim : ARRAY[0..MAX_LAST_ICLA_MOTOR] OF stIclaSim;
END_VAR
```

### Program Logical/Printer/Sim/SimMachine

#### General.st
```iecst
ACTION General:

	FOR iSimIndex:=1 TO MAX_LAST_BLOCK DO
		gTraySim[iSimIndex].Commands.ToIn:=gBlock[iSimIndex].Out.xTrayIn;
		gTraySim[iSimIndex].Commands.ToOut:=gBlock[iSimIndex].Out.xTrayOut;
		gBlock[iSimIndex].In.xTrayIn:=gTraySim[iSimIndex].State.InPosition;
		gBlock[iSimIndex].In.xTrayOut:=gTraySim[iSimIndex].State.OutPosition;
	END_FOR;

	//Signal from the selector
	IF EDGEPOS(gMachine.In.Buttons.xManual) THEN
		gMachine.In.Buttons.xZero:=FALSE;
		gMachine.In.Buttons.xAuto:=FALSE;
	END_IF
	IF EDGEPOS(gMachine.In.Buttons.xZero) THEN
		gMachine.In.Buttons.xManual:=FALSE;
		gMachine.In.Buttons.xAuto:=FALSE;
	END_IF
	IF EDGEPOS(gMachine.In.Buttons.xAuto) THEN
		gMachine.In.Buttons.xManual:=FALSE;
		gMachine.In.Buttons.xZero:=FALSE;
	END_IF

	IF EDGEPOS(gSimMachine.Commands.xToZero) THEN
		gMachine.In.Buttons.xZero:=TRUE;
		gMachine.In.Buttons.xManual:=FALSE;
		gMachine.In.Buttons.xAuto:=FALSE;

		simEventLog.Source := ELOG_TYPE_GENERAL;
		simEventLog.Severity:= ELOG_SEVERITY_INFO;
		simEventLog.Facility:= 0;
		simEventLog.ErrorCode:=0;
		simEventLog.Text := 'Machine going to Zero in Simulation';
		gEventLogLoader(EventData:=ADR(simEventLog));

	END_IF
	IF gSimMachine.Commands.xToZero AND gMachine.St.Mode.xZero THEN
		gSimMachine.Commands.xToZero:=FALSE;
	END_IF

	IF EDGEPOS(gSimMachine.Commands.xToManual) AND gMachine.St.Mode.xManual THEN
		gSimMachine.Commands.xToManual:=FALSE;
	END_IF
	IF EDGEPOS(gSimMachine.Commands.xToManual) THEN
		gMachine.In.Buttons.xZero:=FALSE;
		gMachine.In.Buttons.xManual:=TRUE;
		gMachine.In.Buttons.xAuto:=FALSE;
		gMachine.In.Buttons.xReset:=TRUE;
	END_IF
	IF gSimMachine.Commands.xToManual AND gMachine.St.Mode.xManual THEN
		gSimMachine.Commands.xToManual:=FALSE;
		gMachine.In.Buttons.xReset:=FALSE;
	END_IF

	IF EDGEPOS(gSimMachine.Commands.xToAuto) AND gMachine.St.Mode.xAuto THEN
		gSimMachine.Commands.xToAuto:=FALSE;
	END_IF
	IF EDGEPOS(gSimMachine.Commands.xToAuto) THEN
		gMachine.In.Buttons.xZero:=FALSE;
		gMachine.In.Buttons.xManual:=FALSE;
		gMachine.In.Buttons.xAuto:=TRUE;
		gMachine.In.Buttons.xReset:=TRUE;
	END_IF
	IF gSimMachine.Commands.xToAuto AND gMachine.St.Mode.xAuto THEN
		gSimMachine.Commands.xToAuto:=FALSE;
		gMachine.In.Buttons.xReset:=FALSE;
	END_IF

	IF gSimMachine.Commands.xToProduction THEN
		IF gMachine.Pt.xControlledByLine THEN
			gLine.Commands.Print := TRUE;
		ELSE
			gMachine.commandsSw.xStart_GI := TRUE;
		END_IF
	END_IF
	gSimMachine.Commands.xToProduction := FALSE;

	IF gMachine.Pt.CT.iNumBlocks >= 2 THEN
		ctrlBlock2:=0;
		xBlockExists2:=TRUE;
	ELSE
		ctrlBlock2:=1;
		xBlockExists2:=FALSE;
	END_IF

	//Consent. Doing it more robust. Just allowing this command to speed up simulation
	IF EDGEPOS(gSimMachine.Commands.Consent.xRaiseUpWithNoConsent AND gMachine.St.Consent.xUpWithNoConsentCountingTime) THEN
		gMachine.St.Consent.xUpWithNoConsent := TRUE;
	END_IF

	// Sim feedback clean belt UV position
	IF gMachine.commands.CleanBelt.xPistonFlojet THEN
		gMachine.In.CleanBelt.xLowPosition := FALSE;
		gMachine.In.CleanBelt.xHighPosition := TRUE;
	ELSE
		gMachine.In.CleanBelt.xLowPosition := TRUE;
		gMachine.In.CleanBelt.xHighPosition := FALSE;
	END_IF

END_ACTION
```

#### Initialization.st
```iecst
ACTION Initialization:

	gMachine.In.ProductDetect.pPDSignalSensorL1 := ADR(gSimMachine.Signals.xProductDetectL1);
	gMachine.In.ProductDetect.pPDSignalSensorL2 := ADR(gSimMachine.Signals.xProductDetectL2);
	gMachine.In.ProductDetect.pPDCarriageSignalL1 := ADR(gSimMachine.Signals.xPDCarriageSignalL1);
	gMachine.In.ProductDetect.pPDCarriageSignalL2 := ADR(gSimMachine.Signals.xPDCarriageSignalL2);

	FOR iSimIndex:=1 TO MAX_LAST_BLOCK DO
		gBlock[iSimIndex].In.xAirVenturiOK:=TRUE;
		gBlock[iSimIndex].In.xSiUnitModuleOk:=TRUE;
		gBlock[iSimIndex].In.xDriveProtectionOK:=TRUE;
		gBlock[iSimIndex].In.xDifferentialOK:=TRUE;
		gBlock[iSimIndex].In.Safety.xRearSafetyOK:=TRUE;
		gBlock[iSimIndex].In.Safety.xSafetyOK:=TRUE;
		gBlock[iSimIndex].In.xModuleTemp01Ok:=TRUE;
		gBlock[iSimIndex].In.xModuleTemp02Ok:=TRUE;
		gBlock[iSimIndex].In.xModuleTemp03Ok:=TRUE;
		gBlock[iSimIndex].In.xTrayIn:=TRUE;
		gBlock[iSimIndex].In.Safety.xCurtainEnable01:=TRUE;
		gBlock[iSimIndex].In.Safety.xCurtainEnable02:=TRUE;
		gBlock[iSimIndex].In.Safety.xFrontEStopOK:=TRUE;
		gBlock[iSimIndex].In.Safety.xRearEStopOK:=TRUE;
		gBlock[iSimIndex].In.Safety.xFrontSafetyOK:=TRUE;
		gBlock[iSimIndex].In.xHeaterDcOkBusBar1:=TRUE;
		gBlock[iSimIndex].In.xHeaterDcOkBusBar2:=TRUE;
		FOR iIndexPsu:=1 TO gBlock[iSimIndex].parameters.Hw.iNumHeaterPSU DO
			gBlock[iSimIndex].In.xHeaterDcOkPsu[iIndexPsu]:=TRUE;
			gBlock[iSimIndex].In.xHeaterAcOkPsu[iIndexPsu]:=TRUE;
		END_FOR

		FOR iIndexPsu:=1 TO gBlock[iSimIndex].parameters.Hw.iNumPrintheadsPSU DO
			gBlock[iSimIndex].In.xPrintHeadPSU[iIndexPsu]:=TRUE;
		END_FOR
	END_FOR

	FOR iSimIndex:=1 TO MAX_LAST_BLOCK DO
		gIcla[iSimIndex].Status.xModuleOK:=TRUE;
	END_FOR

	gPhotoCells.status.xBackModuleOk := TRUE;
	gPhotoCells.status.xFrontModuleOk := TRUE;

	gMachine.In.xAirSupply:=TRUE;
	gMachine.In.x24Vdc:=TRUE;

	//We need to write over the permanent var because is loaded during machine init
	//gPermanentBelt.xDriveProtectionOK:=TRUE;
	gBelt.parameters.xDriveProtectionOK:=TRUE;

	webClient.option := httpOPTION_HTTP_11;
	webClient.pHost := ADR(URLHost);
	webClient.pUri := ADR(URIHost);
	webClient.hostPort := 82;
	webClient.method := httpMETHOD_GET;

	webClient.pResponseHeader := ADR(ResponseHeader);
	webClient.pResponseData := ADR(ResponseData);
	webClient.responseDataSize := SIZEOF(ResponseData);
	webClient.pRequestData := ADR(RequestData);
	webClient.requestDataLen := SIZEOF(RequestData);

	gInverterSignalsPowerLink[1].In.ModuleOk := TRUE;
	gInverterSignalsPowerLink[2].In.ModuleOk := TRUE;
	gInverterSignalsPowerLink[3].In.ModuleOk := TRUE;
	gInverterSignalsPowerLink[4].In.ModuleOk := TRUE;
	gInverterSignalsCanOpen[1].In.ModuleOk := TRUE;
	gInverterSignalsCanOpen[2].In.ModuleOk := TRUE;
	gInverterSignalsCanOpen[3].In.ModuleOk := TRUE;
	gInverterSignalsCanOpen[4].In.ModuleOk := TRUE;
	gInverterSignalsPowerLinkABB[1].In.ModuleOk := TRUE;
	gInverterSignalsPowerLinkABB[2].In.ModuleOk := TRUE;
	gInverterSignalsPowerLinkABB[3].In.ModuleOk := TRUE;
	gInverterSignalsPowerLinkABB[4].In.ModuleOk := TRUE;

	gAxisInverter[1].ElecSignals.In.xBreakerOK := TRUE;
	gAxisInverter[2].ElecSignals.In.xBreakerOK := TRUE;
	gAxisInverter[3].ElecSignals.In.xBreakerOK := TRUE;
	gAxisInverter[4].ElecSignals.In.xBreakerOK := TRUE;

	gNonCrash[1].Inputs.xDiffContacOk := TRUE;
	gNonCrash[1].Parameters.DriveUnit.LinealPerimeter.Perimeter:=500;
	gNonCrash[2].Inputs.xDiffContacOk := TRUE;
	gNonCrash[2].Parameters.DriveUnit.LinealPerimeter.Perimeter:=500;

	// ###################################
	// END OF INIT CODE

END_ACTION
```

#### MachineModelCode.st
```iecst
ACTION MachineModelCode:

	//Define the inputs of the Machine depending the machine to Simulate
	CASE gSimMachine.Parameters.MachineType OF
		SIM_MACHINE_2B12BAR:
			gMachine.In.iMachineModelCode:=15;
		SIM_MACHINE_1B6BAR:
			gMachine.In.iMachineModelCode:=51;
		SIM_MACHINE_1B2BAR:
			gMachine.In.iMachineModelCode:=3;
//		SIM_MACHINE_S1400:
//			gMachine.In.iMachineModelCode:=13;
		SIM_MACHINE_S1400_VAC_PWRLNK:
			gMachine.In.iMachineModelCode:=14;
		SIM_MACHINE_S1400_VAC_CAN:
			gMachine.In.iMachineModelCode:=1015;
		SIM_MACHINE_NZ2:
			gMachine.In.iMachineModelCode:=39;
		SIM_MACHINE_NZ2_UV:
			gMachine.In.iMachineModelCode:=40;
		SIM_MACHINE_NZ2_UV_WHITE:
			gMachine.In.iMachineModelCode:=41;
		SIM_MACHINE_CUBE:
			gMachine.In.iMachineModelCode:=10001;
		SIM_MACHINE_CUBE_GULLIVER:
			gMachine.In.iMachineModelCode:=10002;
//		SIM_MACHINE_P5_OIL:
//			gMachine.In.iMachineModelCode:=5;
		SIM_MACHINE_P5_WAT:
			gMachine.In.iMachineModelCode:=6;
		SIM_MACHINE_P4_CBK:
			gMachine.In.iMachineModelCode:=11;
		SIM_MACHINE_MECANO_UV_WHITE:
			gMachine.In.iMachineModelCode:=60;
		SIM_MACHINE_MECANO_UV_OPV:
			gMachine.In.iMachineModelCode:=61;
		SIM_MACHINE_MECANO_UV_WHITE_OPV:
			gMachine.In.iMachineModelCode:=62;
	END_CASE

	//To show or not the second card block layout in diagnostic screen
	CASE  simMachineType OF
		SIM_MACHINE_REAL:
			xShowSecondLayout := FALSE;

		SIM_MACHINE_2B12BAR:

			xShowSecondLayout	:= TRUE;
			xShowThirdLayout	:= TRUE;
			stConfigToShow_Lyout1 := 'P4_PDC_content';
			stConfigToShow_Lyout2 := 'P4_Block1_content';
			stConfigToShow_Lyout3 := 'P4_Block2_content';

		SIM_MACHINE_1B6BAR:
			xShowSecondLayout	:= TRUE;
			xShowThirdLayout	:= FALSE;
			stConfigToShow_Lyout1 := 'P4_PDC_content';
			stConfigToShow_Lyout2 := 'P4_Block1_content';

		SIM_MACHINE_P5_WAT:
			xShowSecondLayout := FALSE;
			xShowThirdLayout	:= FALSE;
			stConfigToShow_Lyout1 := 'P5_S1400_content';
			//stConfigToShow_Lyout2 := 'P4_Block1_content';

		SIM_MACHINE_1B2BAR:
			xShowSecondLayout := FALSE;
			xShowThirdLayout	:= FALSE;
			stConfigToShow_Lyout1 := 'SHIELD_Cards_content';

		SIM_MACHINE_S1400_VAC_PWRLNK,
		SIM_MACHINE_S1400_VAC_CAN:
			xShowSecondLayout := FALSE;
			xShowThirdLayout	:= FALSE;
			stConfigToShow_Lyout1 := 'P5_S1400_content';

		SIM_MACHINE_NZ2,
		SIM_MACHINE_NZ2_UV,
		SIM_MACHINE_NZ2_UV_WHITE:
			xShowSecondLayout := TRUE;
			xShowThirdLayout	:= FALSE;
			stConfigToShow_Lyout1 := 'NZ2_PDC_content';
			stConfigToShow_Lyout2 := 'NZ2_Printer_content';

	ELSE
			xShowSecondLayout	:= FALSE;
			xShowThirdLayout	:= FALSE;
	END_CASE

END_ACTION
```

#### Main.st
```iecst
PROGRAM _INIT

	URLHost := '127.0.0.1';

	Initialization;

	//Call variables to avoid unusefull warnings
	GlobalIO;
	DeviceComms;
	Dryer;
	InkBox;
	Motion;

END_PROGRAM

PROGRAM _CYCLIC

	MachineModelCode;

	General;

	UPS;

	Tests;

	LogTests;

	//Definition of the machine at the end of the code
	IF simMachineTypeEnumCopy<>gSimMachine.Parameters.MachineType THEN
		simMachineType := DINT_TO_INT(gSimMachine.Parameters.MachineType);
		IF simMachineTypeEnumCopy <> SIM_MACHINE_REAL THEN
			xNeedToRestartCPU := TRUE;
		END_IF
	END_IF
	IF simMachineType<>simMachineTypeCopy THEN
		gSimMachine.Parameters.MachineType := simMachineType;
	END_IF

	simMachineTypeCopy := simMachineType;
	simMachineTypeEnumCopy := gSimMachine.Parameters.MachineType;

	//Restart CPU if needed. Done with timer to allow other programs to use the new model and save it before restart
	tonRestart.IN := xNeedToRestartCPU;
	tonRestart.PT := T#300ms;
	tonRestart();
	IF tonRestart.Q THEN
		statusReset := SYSreset(enable:= TRUE, mode:= 2);
	END_IF

END_PROGRAM

PROGRAM _EXIT
	gEventLogManager; //Just here to be able to watch this var
END_PROGRAM
```

#### TestEventLog.st
```iecst
ACTION LogTests:

	IF NOT gSimMachine.Commands.LogTests.xCommand THEN
		RETURN;
	END_IF
	gSimMachine.Commands.LogTests.xCommand := FALSE;

	stEventLogTests.Source := ELOG_TYPE_GENERAL;
	stEventLogTests.Severity:= ELOG_SEVERITY_INFO;
	stEventLogTests.Facility:= 0;
	stEventLogTests.ErrorCode:=0;

	stEventLogTests.Text := 'TEST >>>> ';
	brsstrcat(ADR(stEventLogTests.Text),ADR(gSimMachine.Commands.LogTests.Text));

	gEventLogLoader(EventData := ADR(stEventLogTests));

END_ACTION
```

#### Tests.st
```iecst
ACTION Tests:

	//Configuration of the calling to the TestExecution
	IF xTestPrepareMachine THEN
		URIHost := '/WsTest/PrepareMachine';
	ELSIF xTestPrePrepare THEN
		URIHost := '/WsTest/PrePrepare';
	ELSIF xTestBeltTests THEN
		URIHost := '/WsTest/BeltTests';
	ELSIF xTestConsents THEN
		URIHost := '/WsTest/ConsentTests';
	ELSIF xTestCleaning THEN
		URIHost := '/WsTest/CleaningTests';
	ELSIF xTestLine THEN
		URIHost := '/WsTest/LineTests';
	ELSIF xTestBlock THEN
		URIHost := '/WsTest/BlockTests';
	ELSIF xTestTrVacuum THEN
		URIHost := '/WsTest/TrVacuumTests';
	END_IF

	webClient.enable:=TRUE;
	webClient.send:= xTestPrepareMachine OR xTestPrePrepare OR xTestBeltTests OR xTestConsents OR xTestCleaning OR xTestLine OR xTestBlock OR xTestTrVacuum;
	webClient();

	//Clear Failed and Asserts when starting a new test
	IF EDGEPOS(webClient.send) THEN
		testPassedAsserts:=0;
		testFailedAsserts:=0;
	END_IF

	testMonitor.Enable:=TRUE;
	testMonitor();
	testPassedAsserts:=testMonitor.Informational.PassedAssertCounter;
	testFailedAsserts:=testMonitor.Informational.FailedAssertCounter;
	xSometestFailedAsserts:= testFailedAsserts > 0;

END_ACTION
```

#### UPS.st
```iecst
ACTION UPS:

	gMachine.In.UPSs[1].xLowBattery := gSimMachine.Commands.UPS.xRaiseLowBat;
	gMachine.In.UPSs[1].xPowerFault := gSimMachine.Commands.UPS.xRaisePowerFault;

END_ACTION
```

### Program Logical/Printer/Sim/SimMachine_Fast

#### SimMachine_Fast.var
```iecst
VAR
	Stain : BlinkOnOff;
	tiStainLength : TIME;
	tiStainGap : TIME;
	BoardsFeedMinGap : BlinkOnOff;
	tiBoardTime : TIME;
	tiGapTime : TIME;
	rBeltSpeedMmMs : REAL; (*Belt speed in mm/ms*)
	rPrevStainLength : REAL;
	rPrevStainGap : REAL;
	rPrevBoardLength : REAL;
	rPrevBoardGap : REAL;
	rPrevBeltSpeed : REAL;
	xStainChanged : BOOL;
	xFormatChanged : BOOL;
	xBeltSpeedChanged : BOOL;
	iReasonToContinuousMedia : USINT;
	ExecuteConnect_0 : BOOL;
	SessionConnectInfo_0 : UASessionConnectInfo;
	ConnectionHdl_0 : DWORD;
	UA_Connect_0 : UA_Connect;
	ExecuteGetnamespaceindex_0 : BOOL;
	NamespaceIndex_0 : UINT;
	UA_GetNamespaceIndex_0 : UA_GetNamespaceIndex;
	ExecuteMethodGetHandle_0 : BOOL;
	ObjectNodeID_0 : UANodeID;
	MethodNodeID_0 : UANodeID;
	MethodHdl_0 : DWORD;
	SessionConnectInfo_Energy : UASessionConnectInfo;
	InputArguments_0 : ARRAY[0..9] OF UAMethodArgument;
	OutputArguments_0 : ARRAY[0..9] OF UAMethodArgument;
	UA_MethodGetHandle_0 : UA_MethodGetHandle;
	ExecuteMethodCall_0 : BOOL;
	UA_MethodCall_0 : UA_MethodCall;
	MethodResult_0 : UDINT;
	NewMediaData_0 : stThicknessCtrl_MediaConfig;
	tonNotCallingMethod_0 : TON;
	ExecuteConnect_Energy : BOOL;
	ConnectionHdl_Energy : DWORD;
	UA_Connect_Energy : UA_Connect;
	ExecuteGetnamespaceindex_Energy : BOOL;
	NamespaceIndex_Energy : UINT;
	UA_GetNamespaceIndex_Energy : UA_GetNamespaceIndex;
	ExecuteMethodGetHandle_Energy : BOOL;
	ObjectNodeID_Energy : UANodeID;
	MethodNodeID_Energy : UANodeID;
	MethodHdl_Energy : DWORD;
	InputArguments_Energy : ARRAY[0..9] OF UAMethodArgument;
	OutputArguments_Energy : ARRAY[0..9] OF UAMethodArgument;
	UA_MethodGetHandle_Energy : UA_MethodGetHandle;
	ExecuteMethodCall_Energy : BOOL;
	UA_MethodCall_Energy : UA_MethodCall;
	MethodResult_Energy : UDINT;
	NewMediaData_Energy : stThickCtrl_EnergyMedia;
	tonNotCallingMethod_Energy : TON;
	gDingInputPreviousValue : REAL;
END_VAR
```

#### Media.st
```iecst
ACTION Media:

	IF gThicknessCtrl.status.xNewMediaStackEnabled THEN
		gSimMachine.Parameters.Stack.iMediaQuantityToKeepLoaded := 4;
		gSimMachine.Parameters.Stack.xLoadNewMedia := TRUE;
	END_IF

	IF EDGEPOS(gSimMachine.Commands.Media.xMediaPresent) THEN
		IF gDing.State.xDingInstalled THEN
			gDing.In.rHighDingMm := gSimMachine.Commands.Media.rMediaThickness;
			gDing.In.xDingLow:=TRUE;

		ELSIF gPhotoCells.status.xInstalled THEN
			gPhotoCells.Inputs.Signals.xPhotoCells[1] := TRUE;
		END_IF
		IF gThicknessCtrl.parameters.Detection.ProductDetect.xLoadMedia THEN
			gSimMachine.Signals.xProductDetectL1 := TRUE;
		END_IF
	END_IF

	IF EDGENEG(gSimMachine.Commands.Media.xMediaPresent) THEN
		IF gDing.State.xDingInstalled THEN
			gDing.In.rHighDingMm := 0;
			gDing.In.xDingLow:=FALSE;

		ELSIF gPhotoCells.status.xInstalled THEN
			gPhotoCells.Inputs.Signals.xPhotoCells[1] := FALSE;
		END_IF
		IF gThicknessCtrl.parameters.Detection.ProductDetect.xLoadMedia THEN
			gSimMachine.Signals.xProductDetectL1 := FALSE;
		END_IF
	END_IF

	//Boards entering the printer constantly
	iReasonToContinuousMedia.0 := gSimMachine.Commands.Media.xContinuousMediaPresent;
	iReasonToContinuousMedia.1 := gSimMachine.Commands.Media.xMediaIfFeederFeeding AND gFeeder.Status.CtrlStatus=FEEDERCTRL_FEEDING;
	iReasonToContinuousMedia.2 := gSimMachine.Commands.xStain;

	// Storing previous value
	IF EDGEPOS(iReasonToContinuousMedia > 0 AND gBelt.states.xRuningBelt) THEN
		gDingInputPreviousValue := gDing.In.rHighDingMm;
	END_IF

	xBeltSpeedChanged := rPrevBeltSpeed <> gBelt.states.rCurrentSpeed;
	xFormatChanged := 	rPrevBoardLength <> gMachine.parSw.Media.rLength OR
						rPrevBoardGap <> gMachine.parSw.Media.rGap;
	xStainChanged := 	rPrevStainLength <> gSimMachine.Parameters.rStainLength OR
						rPrevStainGap <> gSimMachine.Parameters.rStainGap;

	IF (xBeltSpeedChanged OR xFormatChanged OR xStainChanged) AND (gBelt.states.rCurrentSpeed > gc_rMinSpeedToStart) THEN
		rBeltSpeedMmMs := (gBelt.states.rCurrentSpeed/60);

		//Board
		tiBoardTime := REAL_TO_TIME(gMachine.parSw.Media.rLength/rBeltSpeedMmMs);
		tiGapTime := REAL_TO_TIME(gMachine.parSw.Media.rGap/rBeltSpeedMmMs);

		//Stain
		tiStainLength := REAL_TO_TIME(gSimMachine.Parameters.rStainLength/rBeltSpeedMmMs);
		tiStainGap := REAL_TO_TIME(gSimMachine.Parameters.rStainGap/rBeltSpeedMmMs);
	END_IF
	rPrevBeltSpeed := gBelt.states.rCurrentSpeed;
	rPrevBoardLength := gMachine.parSw.Media.rLength;
	rPrevBoardGap := gMachine.parSw.Media.rGap;

	//To simulate a media
	BoardsFeedMinGap.tTimeOn := tiBoardTime;
	BoardsFeedMinGap.tTimeOff := tiGapTime;
	BoardsFeedMinGap.xEnable := iReasonToContinuousMedia > 0 AND gBelt.states.xRuningBelt AND NOT gSimMachine.Commands.xStain;
	BoardsFeedMinGap();

	//To simulate a stain over the belt
	Stain.tTimeOn := tiStainLength;
	Stain.tTimeOff := tiStainGap;
	Stain.xEnable := gSimMachine.Commands.xStain;
	Stain();

	IF iReasonToContinuousMedia > 0 AND gBelt.states.xRuningBelt THEN

		IF gDing.State.xDingInstalled THEN
			IF EDGEPOS(BoardsFeedMinGap.xOutput) THEN
				gDing.In.rHighDingMm := gDingInputPreviousValue + gSimMachine.Commands.Media.rMediaThickness;
			ELSIF EDGENEG(BoardsFeedMinGap.xOutput) THEN
				gDing.In.rHighDingMm := gDingInputPreviousValue;
			END_IF
			gDing.In.xDingLow := BoardsFeedMinGap.xOutput OR Stain.xOutput;
			IF gThicknessCtrl.parameters.Detection.ProductDetect.xLoadMedia THEN
				gSimMachine.Signals.xProductDetectL1 := BoardsFeedMinGap.xOutput OR Stain.xOutput;
			END_IF

		ELSIF gPhotoCells.status.xInstalled THEN
			gPhotoCells.Inputs.Signals.xPhotoCells[1] := BoardsFeedMinGap.xOutput;
			IF gThicknessCtrl.parameters.Detection.ProductDetect.xLoadMedia THEN
				gSimMachine.Signals.xProductDetectL1 := BoardsFeedMinGap.xOutput OR Stain.xOutput;
			END_IF
		END_IF

		//Rush proof
		IF gSimMachine.Commands.Media.xRushProof AND EDGEPOS(BoardsFeedMinGap.xOutput) THEN
			gThicknessCtrl.Commands.xRushProof := TRUE;
			//ELSIF NOT BoardsFeedMinGap.xOutput THEN
		ELSIF EDGENEG(gSimMachine.Commands.Media.xRushProof) THEN
			gThicknessCtrl.Commands.xRushProof := FALSE;
		END_IF
	END_IF

	IF EDGEPOS(iReasonToContinuousMedia = 0) THEN
		gDing.In.xDingLow := FALSE;
		gPhotoCells.Inputs.Signals.xPhotoCells[1] := FALSE;
		gSimMachine.Signals.xProductDetectL1 := FALSE;
		gThicknessCtrl.Commands.xRushProof := FALSE;
	END_IF

END_ACTION
```
